KUKA KRL program: EPS_2_25089_SANMH03A_C_20251118074758.src

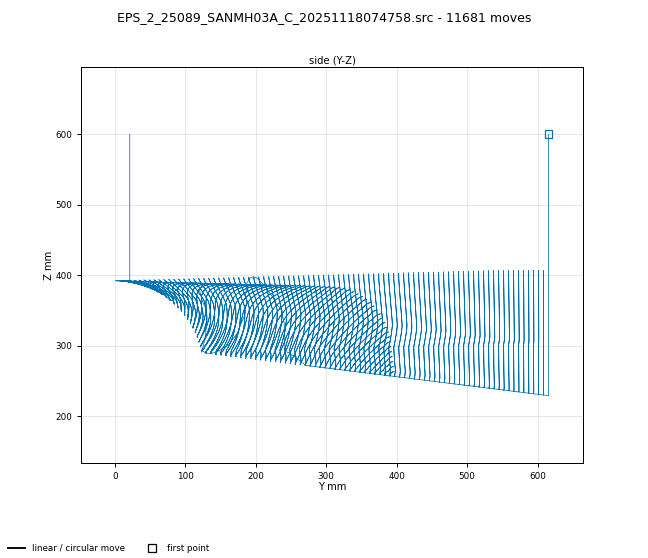
[picture p0: tool path of EPS_2_25089_SANMH03A_C_20251118074758.src, 11681 of 11683 moves have a stored position in this frame; points joined in program order, loops and branches not executed]
&ACCESS RVP
&REL 4
&COMMENT QRS 19112012
&PARAM EDITMASK = *
DEF PART()
EXT BAS (BAS_COMMAND :IN,REAL :IN )
INT I
BAS (#INITMOV,0 )

;KUKA QRS Post kuka4.cps  Date:22-06-2017 !

File_ID=2925

QRS_PRE_INIT()

;Init var - Until changes are made in qrs_pre_init
Outlet_Square_prg=0
Inlet_1_Square_prg=0
Inlet_2_Square_prg=0
Inlet_3_Square_prg=0
Inlet_4_Square_prg=0
Inlet_5_Square_prg=0

Outlet_1={X 0.000, Y 531.880, Z 306.500, B 0.000, E1 0.000 }
Inlet_1={X 0.000, Y 560.070, Z 281.500, B 0.000, E1 180.000 }
Outlet_1_type=201
Inlet_1_type=0
;QRS#1=Sidecore dimensions
;QRS#2=200-8" PVC SDR 35
;QRS#3=DeadEnd 201
;QRS#4=
;QRS#5=
;QRS#6=
;QRS#7=
;QRS#8=
;QRS#9=12-08 PSX
;QRS#10=

;QRS#11=
;QRS#12=
;QRS#13=
;QRS#14=
;QRS#15=
;QRS#16=1220x127x686 2,25'
;QRS#17=EPS Height
;QRS#18=407
;QRS#19=*
;QRS#20= UPDATED VERSION 22-06-2017
;QRS#21=*
Outlet_Square=0100
Inlet_1_Square=00
Inlet_2_Square=0
Inlet_3_Square=0
Inlet_4_Square=0
Inlet_5_Square=0
Mill_Square=1
Outlet_Square_Prg=204
Inlet_1_Square_prg=0

QRS_INIT()

$ADVANCE=5

; T1
PTP {E1 173.634,E2 173.634}
PTP {X 0,Y 615.433,A -85,B 0,C 180,E1 173.634,E2 173.634,E3 0,E4 0,E5 0,E6 0}
QRS_SPEED_INIT()
LIN {X 0,Y 615.433,Z 600,A -85,B 0,C 180,E1 173.634,E2 173.634,E3 0,E4 0,E5 0,E6 0} C_VEL
LIN {X 0,Y 615.433,Z 239.375,A -85,B 0,C 180,E1 173.634,E2 173.634} C_VEL
LIN {X 0,Y 615.433,Z 231.198,A -85,B 0,C 180,E1 173.634,E2 173.634} C_VEL
LIN {X 0,Y 615.441,Z 229.198,A -85,B 0,C 180,E1 173.448,E2 173.448} C_VEL
LIN {X 0,Y 615.497,Z 229.194,A -85,B 0,C 180,E1 170.806,E2 170.806} C_VEL
LIN {X 0,Y 615.433,Z 229.195,A -85,B 0,C 180,E1 168.143,E2 168.143} C_VEL
LIN {X 0,Y 615.431,Z 229.196,A -85,B 0,C 180,E1 166.083,E2 166.083} C_VEL
LIN {X 0,Y 615.468,Z 229.199,A -85,B 0,C 180,E1 163.418,E2 163.418} C_VEL
LIN {X 0,Y 615.454,Z 229.194,A -85,B 0,C 180,E1 160.666,E2 160.666} C_VEL
LIN {X 0,Y 615.441,Z 229.195,A -85,B 0,C 180,E1 158.572,E2 158.572} C_VEL
LIN {X 0,Y 615.432,Z 229.196,A -85,B 0,C 180,E1 156.447,E2 156.447} C_VEL
LIN {X 0,Y 615.428,Z 229.197,A -85,B 0,C 180,E1 154.288,E2 154.288} C_VEL
LIN {X 0,Y 615.484,Z 229.201,A -85,B 0,C 180,E1 151.548,E2 151.548} C_VEL
LIN {X 0,Y 615.446,Z 229.195,A -85,B 0,C 180,E1 148.918,E2 148.918} C_VEL
LIN {X 0,Y 615.426,Z 229.197,A -85,B 0,C 180,E1 146.472,E2 146.472} C_VEL
LIN {X 0,Y 615.44,Z 229.198,A -85,B 0,C 180,E1 144.17,E2 144.17} C_VEL
LIN {X 0,Y 615.468,Z 229.199,A -85,B 0,C 180,E1 141.938,E2 141.938} C_VEL
LIN {X 0,Y 615.468,Z 229.195,A -85,B 0,C 180,E1 139.4,E2 139.4} C_VEL
LIN {X 0,Y 615.427,Z 229.197,A -85,B 0,C 180,E1 136.957,E2 136.957} C_VEL
LIN {X 0,Y 615.424,Z 229.197,A -85,B 0,C 180,E1 134.935,E2 134.935} C_VEL
LIN {X 0,Y 615.448,Z 229.199,A -85,B 0,C 180,E1 132.355,E2 132.355} C_VEL
LIN {X 0,Y 615.475,Z 229.197,A -85,B 0,C 180,E1 129.75,E2 129.75} C_VEL
LIN {X 0,Y 615.426,Z 229.197,A -85,B 0,C 180,E1 127.245,E2 127.245} C_VEL
LIN {X 0,Y 615.434,Z 229.199,A -85,B 0,C 180,E1 124.705,E2 124.705} C_VEL
LIN {X 0,Y 615.478,Z 229.2,A -85,B 0,C 180,E1 122.342,E2 122.342} C_VEL
LIN {X 0,Y 615.45,Z 229.197,A -85,B 0,C 180,E1 119.802,E2 119.802} C_VEL
LIN {X 0,Y 615.452,Z 229.198,A -85,B 0,C 180,E1 117.916,E2 117.916} C_VEL
LIN {X 0,Y 615.423,Z 229.198,A -85,B 0,C 180,E1 115.572,E2 115.572} C_VEL
LIN {X 0,Y 615.419,Z 229.199,A -85,B 0,C 180,E1 113.559,E2 113.559} C_VEL
LIN {X 0,Y 615.416,Z 229.199,A -85,B 0,C 180,E1 111.434,E2 111.434} C_VEL
LIN {X 0,Y 615.419,Z 229.199,A -85,B 0,C 180,E1 109.34,E2 109.34} C_VEL
LIN {X 0,Y 615.474,Z 229.201,A -85,B 0,C 180,E1 106.452,E2 106.452} C_VEL
LIN {X 0,Y 615.419,Z 229.199,A -85,B 0,C 180,E1 103.875,E2 103.875} C_VEL
LIN {X 0,Y 615.415,Z 229.2,A -85,B 0,C 180,E1 101.862,E2 101.862} C_VEL
LIN {X 0,Y 615.416,Z 229.199,A -85,B 0,C 180,E1 99.863,E2 99.863} C_VEL
LIN {X 0,Y 615.414,Z 229.199,A -85,B 0,C 180,E1 97.876,E2 97.876} C_VEL
LIN {X 0,Y 615.414,Z 229.2,A -85,B 0,C 180,E1 95.899,E2 95.899} C_VEL
LIN {X 0,Y 615.449,Z 229.2,A -85,B 0,C 180,E1 93.273,E2 93.273} C_VEL
LIN {X 0,Y 615.452,Z 229.2,A -85,B 0,C 180,E1 90.654,E2 90.654} C_VEL
LIN {X 0,Y 615.412,Z 229.2,A -85,B 0,C 180,E1 88.037,E2 88.037} C_VEL
LIN {X 0,Y 615.457,Z 229.2,A -85,B 0,C 180,E1 85.415,E2 85.415} C_VEL
LIN {X 0,Y 615.445,Z 229.2,A -85,B 0,C 180,E1 82.784,E2 82.784} C_VEL
LIN {X 0,Y 615.416,Z 229.199,A -85,B 0,C 180,E1 80.137,E2 80.137} C_VEL
LIN {X 0,Y 615.477,Z 229.2,A -85,B 0,C 180,E1 77.47,E2 77.47} C_VEL
LIN {X 0,Y 615.428,Z 229.199,A -85,B 0,C 180,E1 74.773,E2 74.773} C_VEL
LIN {X 0,Y 615.423,Z 229.199,A -85,B 0,C 180,E1 72.728,E2 72.728} C_VEL
LIN {X 0,Y 615.419,Z 229.199,A -85,B 0,C 180,E1 70.66,E2 70.66} C_VEL
LIN {X 0,Y 615.416,Z 229.199,A -85,B 0,C 180,E1 68.566,E2 68.566} C_VEL
LIN {X 0,Y 615.419,Z 229.199,A -85,B 0,C 180,E1 66.442,E2 66.442} C_VEL
LIN {X 0,Y 615.484,Z 229.2,A -85,B 0,C 180,E1 63.556,E2 63.556} C_VEL
LIN {X 0,Y 615.45,Z 229.199,A -85,B 0,C 180,E1 61.341,E2 61.341} C_VEL
LIN {X 0,Y 615.42,Z 229.198,A -85,B 0,C 180,E1 58.911,E2 58.911} C_VEL
LIN {X 0,Y 615.434,Z 229.198,A -85,B 0,C 180,E1 56.461,E2 56.461} C_VEL
LIN {X 0,Y 615.455,Z 229.199,A -85,B 0,C 180,E1 53.574,E2 53.574} C_VEL
LIN {X 0,Y 615.422,Z 229.198,A -85,B 0,C 180,E1 50.935,E2 50.935} C_VEL
LIN {X 0,Y 615.451,Z 229.196,A -85,B 0,C 180,E1 48.524,E2 48.524} C_VEL
LIN {X 0,Y 615.465,Z 229.199,A -85,B 0,C 180,E1 45.85,E2 45.85} C_VEL
LIN {X 0,Y 615.479,Z 229.2,A -85,B 0,C 180,E1 43.998,E2 43.998} C_VEL
LIN {X 0,Y 615.427,Z 229.198,A -85,B 0,C 180,E1 41.471,E2 41.471} C_VEL
LIN {X 0,Y 615.442,Z 229.196,A -85,B 0,C 180,E1 38.9,E2 38.9} C_VEL
LIN {X 0,Y 615.482,Z 229.201,A -85,B 0,C 180,E1 36.418,E2 36.418} C_VEL
LIN {X 0,Y 615.452,Z 229.199,A -85,B 0,C 180,E1 34.017,E2 34.017} C_VEL
LIN {X 0,Y 615.428,Z 229.197,A -85,B 0,C 180,E1 31.682,E2 31.682} C_VEL
LIN {X 0,Y 615.428,Z 229.196,A -85,B 0,C 180,E1 29.403,E2 29.403} C_VEL
LIN {X 0,Y 615.457,Z 229.195,A -85,B 0,C 180,E1 27.042,E2 27.042} C_VEL
LIN {X 0,Y 615.454,Z 229.199,A -85,B 0,C 180,E1 24.268,E2 24.268} C_VEL
LIN {X 0,Y 615.439,Z 229.198,A -85,B 0,C 180,E1 22.133,E2 22.133} C_VEL
LIN {X 0,Y 615.432,Z 229.197,A -85,B 0,C 180,E1 20.029,E2 20.029} C_VEL
LIN {X 0,Y 615.43,Z 229.196,A -85,B 0,C 180,E1 17.953,E2 17.953} C_VEL
LIN {X 0,Y 615.48,Z 229.193,A -85,B 0,C 180,E1 15.221,E2 15.221} C_VEL
LIN {X 0,Y 615.451,Z 229.198,A -85,B 0,C 180,E1 12.526,E2 12.526} C_VEL
LIN {X 0,Y 615.447,Z 229.198,A -85,B 0,C 180,E1 10.523,E2 10.523} C_VEL
LIN {X 0,Y 615.445,Z 229.198,A -85,B 0,C 180,E1 8.533,E2 8.533} C_VEL
LIN {X 0,Y 615.444,Z 229.197,A -85,B 0,C 180,E1 6.553,E2 6.553} C_VEL
LIN {X 0,Y 615.443,Z 229.197,A -85,B 0,C 180,E1 4.581,E2 4.581} C_VEL
LIN {X 0,Y 615.441,Z 229.197,A -85,B 0,C 180,E1 2.614,E2 2.614} C_VEL
LIN {X 0,Y 615.441,Z 229.197,A -85,B 0,C 180,E1 0.65,E2 0.65} C_VEL
LIN {X 0,Y 615.441,Z 229.197,A -85,B 0,C 180,E1 -1.312,E2 -1.312} C_VEL
LIN {X 0,Y 615.441,Z 229.197,A -85,B 0,C 180,E1 -3.277,E2 -3.277} C_VEL
LIN {X 0,Y 615.44,Z 229.197,A -85,B 0,C 180,E1 -5.245,E2 -5.245} C_VEL
LIN {X 0,Y 615.44,Z 229.196,A -85,B 0,C 180,E1 -7.22,E2 -7.22} C_VEL
LIN {X 0,Y 615.439,Z 229.196,A -85,B 0,C 180,E1 -9.203,E2 -9.203} C_VEL
LIN {X 0,Y 615.438,Z 229.196,A -85,B 0,C 180,E1 -11.197,E2 -11.197} C_VEL
LIN {X 0,Y 615.469,Z 229.191,A -85,B 0,C 180,E1 -13.878,E2 -13.878} C_VEL
LIN {X 0,Y 615.468,Z 229.199,A -85,B 0,C 180,E1 -16.59,E2 -16.59} C_VEL
LIN {X 0,Y 615.457,Z 229.198,A -85,B 0,C 180,E1 -18.65,E2 -18.65} C_VEL
LIN {X 0,Y 615.449,Z 229.197,A -85,B 0,C 180,E1 -20.735,E2 -20.735} C_VEL
LIN {X 0,Y 615.442,Z 229.196,A -85,B 0,C 180,E1 -22.849,E2 -22.849} C_VEL
LIN {X 0,Y 615.439,Z 229.194,A -85,B 0,C 180,E1 -24.996,E2 -24.996} C_VEL
LIN {X 0,Y 615.496,Z 229.195,A -85,B 0,C 180,E1 -27.917,E2 -27.917} C_VEL
LIN {X 0,Y 615.481,Z 229.199,A -85,B 0,C 180,E1 -30.163,E2 -30.163} C_VEL
LIN {X 0,Y 615.45,Z 229.196,A -85,B 0,C 180,E1 -32.462,E2 -32.462} C_VEL
LIN {X 0,Y 615.439,Z 229.194,A -85,B 0,C 180,E1 -34.82,E2 -34.82} C_VEL
LIN {X 0,Y 615.473,Z 229.189,A -85,B 0,C 180,E1 -37.245,E2 -37.245} C_VEL
LIN {X 0,Y 615.464,Z 229.198,A -85,B 0,C 180,E1 -40.088,E2 -40.088} C_VEL
LIN {X 0,Y 615.444,Z 229.195,A -85,B 0,C 180,E1 -42.359,E2 -42.359} C_VEL
LIN {X 0,Y 615.471,Z 229.19,A -85,B 0,C 180,E1 -45.072,E2 -45.072} C_VEL
LIN {X 0,Y 615.468,Z 229.19,A -85,B 0,C 180,E1 -46.956,E2 -46.956} C_VEL
LIN {X 0,Y 615.491,Z 229.616,A -85,B 0,C 180,E1 -47.649,E2 -47.649} C_VEL
LIN {X 0,Y 615.439,Z 234.214,A -85,B 0,C 180,E1 -50.247,E2 -50.247} C_VEL
LIN {X 0,Y 615.494,Z 238.966,A -85,B 0,C 180,E1 -52.759,E2 -52.759} C_VEL
LIN {X 0,Y 615.486,Z 244.106,A -85,B 0,C 180,E1 -55.301,E2 -55.301} C_VEL
LIN {X 0,Y 615.472,Z 249.184,A -85,B 0,C 180,E1 -57.673,E2 -57.673} C_VEL
LIN {X 0,Y 615.449,Z 254.91,A -85,B 0,C 180,E1 -60.213,E2 -60.213} C_VEL
LIN {X 0,Y 615.475,Z 261.498,A -85,B 0,C 180,E1 -62.959,E2 -62.959} C_VEL
LIN {X 0,Y 615.47,Z 266.533,A -85,B 0,C 180,E1 -65.008,E2 -65.008} C_VEL
LIN {X 0,Y 615.475,Z 273.166,A -85,B 0,C 180,E1 -67.658,E2 -67.658} C_VEL
LIN {X 0,Y 615.484,Z 279.039,A -85,B 0,C 180,E1 -69.968,E2 -69.968} C_VEL
LIN {X 0,Y 615.488,Z 286.193,A -85,B 0,C 180,E1 -72.73,E2 -72.73} C_VEL
LIN {X 0,Y 615.466,Z 293.325,A -85,B 0,C 180,E1 -75.451,E2 -75.451} C_VEL
LIN {X 0,Y 615.478,Z 300.472,A -85,B 0,C 180,E1 -78.139,E2 -78.139} C_VEL
LIN {X 0,Y 615.498,Z 301.076,A -85,B 0,C 180,E1 -78.369,E2 -78.369} C_VEL
LIN {X 0,Y 615.485,Z 316.87,A -85,B 0,C 180,E1 -78.724,E2 -78.724} C_VEL
LIN {X 0,Y 615.445,Z 329.215,A -85,B 0,C 180,E1 -79.134,E2 -79.134} C_VEL
LIN {X 0,Y 615.44,Z 340.49,A -85,B 0,C 180,E1 -79.639,E2 -79.639} C_VEL
LIN {X 0,Y 615.49,Z 351.998,A -85,B 0,C 180,E1 -80.304,E2 -80.304} C_VEL
LIN {X 0,Y 615.499,Z 362.344,A -85,B 0,C 180,E1 -81.05,E2 -81.05} C_VEL
LIN {X 0,Y 615.497,Z 370.814,A -85,B 0,C 180,E1 -81.794,E2 -81.794} C_VEL
LIN {X 0,Y 615.498,Z 378.608,A -85,B 0,C 180,E1 -82.62,E2 -82.62} C_VEL
LIN {X 0,Y 615.496,Z 386.204,A -85,B 0,C 180,E1 -83.608,E2 -83.608} C_VEL
LIN {X 0,Y 615.498,Z 393.205,A -85,B 0,C 180,E1 -84.759,E2 -84.759} C_VEL
LIN {X 0,Y 615.494,Z 397.852,A -85,B 0,C 180,E1 -85.744,E2 -85.744} C_VEL
LIN {X 0,Y 615.494,Z 401.399,A -85,B 0,C 180,E1 -86.727,E2 -86.727} C_VEL
LIN {X 0,Y 615.497,Z 403.233,A -85,B 0,C 180,E1 -87.382,E2 -87.382} C_VEL
LIN {X 0,Y 615.5,Z 404.608,A -85,B 0,C 180,E1 -88.037,E2 -88.037} C_VEL
LIN {X 0,Y 615.496,Z 406.173,A -85,B 0,C 180,E1 -89.346,E2 -89.346} C_VEL
LIN {X 0,Y 615.494,Z 406.389,A -85,B 0,C 180,E1 -90,E2 -90} C_VEL
LIN {X 0,Y 615.495,Z 405.58,A -85,B 0,C 180,E1 -91.309,E2 -91.309} C_VEL
LIN {X 0,Y 615.5,Z 404.608,A -85,B 0,C 180,E1 -91.963,E2 -91.963} C_VEL
LIN {X 0,Y 615.497,Z 403.233,A -85,B 0,C 180,E1 -92.618,E2 -92.618} C_VEL
LIN {X 0,Y 615.496,Z 400.35,A -85,B 0,C 180,E1 -93.601,E2 -93.601} C_VEL
LIN {X 0,Y 615.498,Z 396.442,A -85,B 0,C 180,E1 -94.584,E2 -94.584} C_VEL
LIN {X 0,Y 615.499,Z 391.406,A -85,B 0,C 180,E1 -95.57,E2 -95.57} C_VEL
LIN {X 0,Y 615.497,Z 384.875,A -85,B 0,C 180,E1 -96.583,E2 -96.583} C_VEL
LIN {X 0,Y 615.497,Z 377.135,A -85,B 0,C 180,E1 -97.545,E2 -97.545} C_VEL
LIN {X 0,Y 615.498,Z 369.047,A -85,B 0,C 180,E1 -98.371,E2 -98.371} C_VEL
LIN {X 0,Y 615.499,Z 359.17,A -85,B 0,C 180,E1 -99.198,E2 -99.198} C_VEL
LIN {X 0,Y 615.472,Z 347.988,A -85,B 0,C 180,E1 -99.945,E2 -99.945} C_VEL
LIN {X 0,Y 615.437,Z 337.036,A -85,B 0,C 180,E1 -100.528,E2 -100.528} C_VEL
LIN {X 0,Y 615.457,Z 324.807,A -85,B 0,C 180,E1 -101.029,E2 -101.029} C_VEL
LIN {X 0,Y 615.499,Z 312.075,A -85,B 0,C 180,E1 -101.401,E2 -101.401} C_VEL
LIN {X 0,Y 615.498,Z 301.076,A -85,B 0,C 180,E1 -101.631,E2 -101.631} C_VEL
LIN {X 0,Y 615.471,Z 294.981,A -85,B 0,C 180,E1 -103.925,E2 -103.925} C_VEL
LIN {X 0,Y 615.486,Z 287.968,A -85,B 0,C 180,E1 -106.586,E2 -106.586} C_VEL
LIN {X 0,Y 615.484,Z 280.83,A -85,B 0,C 180,E1 -109.338,E2 -109.338} C_VEL
LIN {X 0,Y 615.494,Z 273.68,A -85,B 0,C 180,E1 -112.136,E2 -112.136} C_VEL
LIN {X 0,Y 615.467,Z 268.326,A -85,B 0,C 180,E1 -114.272,E2 -114.272} C_VEL
LIN {X 0,Y 615.446,Z 262.964,A -85,B 0,C 180,E1 -116.445,E2 -116.445} C_VEL
LIN {X 0,Y 615.48,Z 255.804,A -85,B 0,C 180,E1 -119.406,E2 -119.406} C_VEL
LIN {X 0,Y 615.454,Z 250.603,A -85,B 0,C 180,E1 -121.686,E2 -121.686} C_VEL
LIN {X 0,Y 615.484,Z 245.53,A -85,B 0,C 180,E1 -124.021,E2 -124.021} C_VEL
LIN {X 0,Y 615.469,Z 240.585,A -85,B 0,C 180,E1 -126.425,E2 -126.425} C_VEL
LIN {X 0,Y 615.499,Z 235.479,A -85,B 0,C 180,E1 -129.062,E2 -129.062} C_VEL
LIN {X 0,Y 615.447,Z 231.131,A -85,B 0,C 180,E1 -131.476,E2 -131.476} C_VEL
LIN {X 0,Y 615.491,Z 229.616,A -85,B 0,C 180,E1 -132.351,E2 -132.351} C_VEL
LIN {X 0,Y 615.452,Z 229.191,A -85,B 0,C 180,E1 -133.246,E2 -133.246} C_VEL
LIN {X 0,Y 615.462,Z 229.198,A -85,B 0,C 180,E1 -136.004,E2 -136.004} C_VEL
LIN {X 0,Y 615.469,Z 229.19,A -85,B 0,C 180,E1 -138.906,E2 -138.906} C_VEL
LIN {X 0,Y 615.449,Z 229.192,A -85,B 0,C 180,E1 -141.091,E2 -141.091} C_VEL
LIN {X 0,Y 615.447,Z 229.196,A -85,B 0,C 180,E1 -143.57,E2 -143.57} C_VEL
LIN {X 0,Y 615.493,Z 229.189,A -85,B 0,C 180,E1 -146.463,E2 -146.463} C_VEL
LIN {X 0,Y 615.441,Z 229.193,A -85,B 0,C 180,E1 -149.075,E2 -149.075} C_VEL
LIN {X 0,Y 615.457,Z 229.197,A -85,B 0,C 180,E1 -151.552,E2 -151.552} C_VEL
LIN {X 0,Y 615.472,Z 229.19,A -85,B 0,C 180,E1 -154.431,E2 -154.431} C_VEL
LIN {X 0,Y 615.465,Z 229.191,A -85,B 0,C 180,E1 -156.44,E2 -156.44} C_VEL
LIN {X 0,Y 615.45,Z 229.192,A -85,B 0,C 180,E1 -158.564,E2 -158.564} C_VEL
LIN {X 0,Y 615.441,Z 229.193,A -85,B 0,C 180,E1 -160.658,E2 -160.658} C_VEL
LIN {X 0,Y 615.437,Z 229.194,A -85,B 0,C 180,E1 -162.725,E2 -162.725} C_VEL
LIN {X 0,Y 615.48,Z 229.199,A -85,B 0,C 180,E1 -165.448,E2 -165.448} C_VEL
LIN {X 0,Y 615.463,Z 229.192,A -85,B 0,C 180,E1 -168.136,E2 -168.136} C_VEL
LIN {X 0,Y 615.457,Z 229.192,A -85,B 0,C 180,E1 -170.134,E2 -170.134} C_VEL
LIN {X 0,Y 615.454,Z 229.192,A -85,B 0,C 180,E1 -172.121,E2 -172.121} C_VEL
LIN {X 0,Y 615.451,Z 229.193,A -85,B 0,C 180,E1 -174.098,E2 -174.098} C_VEL
LIN {X 0,Y 615.449,Z 229.193,A -85,B 0,C 180,E1 -176.068,E2 -176.068} C_VEL
LIN {X 0,Y 615.447,Z 229.193,A -85,B 0,C 180,E1 -178.033,E2 -178.033} C_VEL
LIN {X 0,Y 615.446,Z 229.193,A -85,B 0,C 180,E1 -179.996,E2 -179.996} C_VEL
LIN {X 0,Y 615.444,Z 229.194,A -85,B 0,C 180,E1 -181.959,E2 -181.959} C_VEL
LIN {X 0,Y 615.443,Z 229.194,A -85,B 0,C 180,E1 -183.925,E2 -183.925} C_VEL
LIN {X 0,Y 615.441,Z 229.194,A -85,B 0,C 180,E1 -185.895,E2 -185.895} C_VEL
LIN {X 0,Y 615.441,Z 229.198,A -85,B 0,C 180,E1 -186.552,E2 -186.552} C_VEL
LIN {X 0,Y 614.816,Z 229.343,A -85,B 0,C 180,E1 -187.098,E2 -187.098} C_VEL
LIN {X 0,Y 612.019,Z 229.743,A -85,B 0,C 180,E1 -187.984,E2 -187.984} C_VEL
LIN {X 0,Y 609.616,Z 230.058,A -85,B 0,C 180,E1 -188.697,E2 -188.697} C_VEL
LIN {X 0,Y 608.553,Z 230.181,A -85,B 0,C 180,E1 -189.246,E2 -189.246} C_VEL
LIN {X 0,Y 608.45,Z 230.191,A -85,B 0,C 180,E1 -189.432,E2 -189.432} C_VEL
LIN {X 0,Y 608.416,Z 230.192,A -85,B 0,C 180,E1 -191.996,E2 -191.996} C_VEL
LIN {X 0,Y 608.452,Z 230.195,A -85,B 0,C 180,E1 -194.716,E2 -194.716} C_VEL
LIN {X 0,Y 608.422,Z 230.193,A -85,B 0,C 180,E1 -197.472,E2 -197.472} C_VEL
LIN {X 0,Y 608.413,Z 230.193,A -85,B 0,C 180,E1 -199.567,E2 -199.567} C_VEL
LIN {X 0,Y 608.424,Z 230.191,A -85,B 0,C 180,E1 -201.688,E2 -201.688} C_VEL
LIN {X 0,Y 608.428,Z 230.2,A -85,B 0,C 180,E1 -204.566,E2 -204.566} C_VEL
LIN {X 0,Y 608.407,Z 230.193,A -85,B 0,C 180,E1 -207.514,E2 -207.514} C_VEL
LIN {X 0,Y 608.419,Z 230.194,A -85,B 0,C 180,E1 -209.966,E2 -209.966} C_VEL
LIN {X 0,Y 608.429,Z 230.194,A -85,B 0,C 180,E1 -212.874,E2 -212.874} C_VEL
LIN {X 0,Y 608.399,Z 230.194,A -85,B 0,C 180,E1 -215.273,E2 -215.273} C_VEL
LIN {X 0,Y 608.441,Z 230.199,A -85,B 0,C 180,E1 -218.239,E2 -218.239} C_VEL
LIN {X 0,Y 608.464,Z 230.195,A -85,B 0,C 180,E1 -220.332,E2 -220.332} C_VEL
LIN {X 0,Y 608.402,Z 230.194,A -85,B 0,C 180,E1 -222.956,E2 -222.956} C_VEL
LIN {X 0,Y 608.399,Z 230.194,A -85,B 0,C 180,E1 -225.2,E2 -225.2} C_VEL
LIN {X 0,Y 608.454,Z 230.196,A -85,B 0,C 180,E1 -227.939,E2 -227.939} C_VEL
LIN {X 0,Y 608.424,Z 230.192,A -85,B 0,C 180,E1 -230.697,E2 -230.697} C_VEL
LIN {X 0,Y 608.393,Z 230.195,A -85,B 0,C 180,E1 -233.082,E2 -233.082} C_VEL
LIN {X 0,Y 608.433,Z 230.195,A -85,B 0,C 180,E1 -235.529,E2 -235.529} C_VEL
LIN {X 0,Y 608.443,Z 230.197,A -85,B 0,C 180,E1 -237.905,E2 -237.905} C_VEL
LIN {X 0,Y 608.432,Z 230.193,A -85,B 0,C 180,E1 -240.219,E2 -240.219} C_VEL
LIN {X 0,Y 608.412,Z 230.193,A -85,B 0,C 180,E1 -242.79,E2 -242.79} C_VEL
LIN {X 0,Y 608.45,Z 230.194,A -85,B 0,C 180,E1 -245.836,E2 -245.836} C_VEL
LIN {X 0,Y 608.415,Z 230.193,A -85,B 0,C 180,E1 -248.307,E2 -248.307} C_VEL
LIN {X 0,Y 608.435,Z 230.195,A -85,B 0,C 180,E1 -251.13,E2 -251.13} C_VEL
LIN {X 0,Y 608.416,Z 230.195,A -85,B 0,C 180,E1 -253.905,E2 -253.905} C_VEL
LIN {X 0,Y 608.401,Z 230.195,A -85,B 0,C 180,E1 -255.979,E2 -255.979} C_VEL
LIN {X 0,Y 608.402,Z 230.195,A -85,B 0,C 180,E1 -257.999,E2 -257.999} C_VEL
LIN {X 0,Y 608.395,Z 230.195,A -85,B 0,C 180,E1 -260.022,E2 -260.022} C_VEL
LIN {X 0,Y 608.412,Z 230.193,A -85,B 0,C 180,E1 -262.032,E2 -262.032} C_VEL
LIN {X 0,Y 608.422,Z 230.195,A -85,B 0,C 180,E1 -264.698,E2 -264.698} C_VEL
LIN {X 0,Y 608.442,Z 230.195,A -85,B 0,C 180,E1 -267.352,E2 -267.352} C_VEL
LIN {X 0,Y 608.403,Z 230.194,A -85,B 0,C 180,E1 -270,E2 -270} C_VEL
LIN {X 0,Y 608.442,Z 230.195,A -85,B 0,C 180,E1 -272.648,E2 -272.648} C_VEL
LIN {X 0,Y 608.422,Z 230.195,A -85,B 0,C 180,E1 -275.302,E2 -275.302} C_VEL
LIN {X 0,Y 608.412,Z 230.193,A -85,B 0,C 180,E1 -277.968,E2 -277.968} C_VEL
LIN {X 0,Y 608.444,Z 230.198,A -85,B 0,C 180,E1 -280.65,E2 -280.65} C_VEL
LIN {X 0,Y 608.405,Z 230.195,A -85,B 0,C 180,E1 -283.357,E2 -283.357} C_VEL
LIN {X 0,Y 608.411,Z 230.193,A -85,B 0,C 180,E1 -285.407,E2 -285.407} C_VEL
LIN {X 0,Y 608.391,Z 230.195,A -85,B 0,C 180,E1 -287.478,E2 -287.478} C_VEL
LIN {X 0,Y 608.392,Z 230.195,A -85,B 0,C 180,E1 -289.572,E2 -289.572} C_VEL
LIN {X 0,Y 608.48,Z 230.194,A -85,B 0,C 180,E1 -292.405,E2 -292.405} C_VEL
LIN {X 0,Y 608.42,Z 230.199,A -85,B 0,C 180,E1 -294.572,E2 -294.572} C_VEL
LIN {X 0,Y 608.412,Z 230.193,A -85,B 0,C 180,E1 -297.21,E2 -297.21} C_VEL
LIN {X 0,Y 608.464,Z 230.192,A -85,B 0,C 180,E1 -299.985,E2 -299.985} C_VEL
LIN {X 0,Y 608.407,Z 230.194,A -85,B 0,C 180,E1 -302.882,E2 -302.882} C_VEL
LIN {X 0,Y 608.396,Z 230.195,A -85,B 0,C 180,E1 -305.28,E2 -305.28} C_VEL
LIN {X 0,Y 608.444,Z 230.196,A -85,B 0,C 180,E1 -308.248,E2 -308.248} C_VEL
LIN {X 0,Y 608.425,Z 230.196,A -85,B 0,C 180,E1 -310.336,E2 -310.336} C_VEL
LIN {X 0,Y 608.395,Z 230.195,A -85,B 0,C 180,E1 -312.964,E2 -312.964} C_VEL
LIN {X 0,Y 608.452,Z 230.196,A -85,B 0,C 180,E1 -315.735,E2 -315.735} C_VEL
LIN {X 0,Y 608.459,Z 230.195,A -85,B 0,C 180,E1 -317.947,E2 -317.947} C_VEL
LIN {X 0,Y 608.397,Z 230.195,A -85,B 0,C 180,E1 -320.563,E2 -320.563} C_VEL
LIN {X 0,Y 608.416,Z 230.194,A -85,B 0,C 180,E1 -323.09,E2 -323.09} C_VEL
LIN {X 0,Y 608.45,Z 230.197,A -85,B 0,C 180,E1 -325.537,E2 -325.537} C_VEL
LIN {X 0,Y 608.444,Z 230.193,A -85,B 0,C 180,E1 -327.911,E2 -327.911} C_VEL
LIN {X 0,Y 608.414,Z 230.193,A -85,B 0,C 180,E1 -330.224,E2 -330.224} C_VEL
LIN {X 0,Y 608.441,Z 230.19,A -85,B 0,C 180,E1 -332.797,E2 -332.797} C_VEL
LIN {X 0,Y 608.435,Z 230.193,A -85,B 0,C 180,E1 -335.853,E2 -335.853} C_VEL
LIN {X 0,Y 608.424,Z 230.191,A -85,B 0,C 180,E1 -338.312,E2 -338.312} C_VEL
LIN {X 0,Y 608.434,Z 230.199,A -85,B 0,C 180,E1 -341.135,E2 -341.135} C_VEL
LIN {X 0,Y 608.414,Z 230.193,A -85,B 0,C 180,E1 -343.91,E2 -343.91} C_VEL
LIN {X 0,Y 608.451,Z 230.191,A -85,B 0,C 180,E1 -346.648,E2 -346.648} C_VEL
LIN {X 0,Y 608.438,Z 230.194,A -85,B 0,C 180,E1 -349.354,E2 -349.354} C_VEL
LIN {X 0,Y 608.425,Z 230.195,A -85,B 0,C 180,E1 -351.368,E2 -351.368} C_VEL
LIN {X 0,Y 608.42,Z 230.195,A -85,B 0,C 180,E1 -353.404,E2 -353.404} C_VEL
LIN {X 0,Y 608.415,Z 230.195,A -85,B 0,C 180,E1 -355.366,E2 -355.366} C_VEL
LIN {X 0,Y 608.437,Z 230.192,A -85,B 0,C 180,E1 -357.356,E2 -357.356} C_VEL
LIN {X 0,Y 608.439,Z 230.19,A -85,B 0,C 180,E1 -360.004,E2 -360.004} C_VEL
LIN {X 0,Y 608.48,Z 230.194,A -85,B 0,C 180,E1 -362.652,E2 -362.652} C_VEL
LIN {X 0,Y 608.423,Z 230.192,A -85,B 0,C 180,E1 -365.306,E2 -365.306} C_VEL
LIN {X 0,Y 608.413,Z 230.193,A -85,B 0,C 180,E1 -367.303,E2 -367.303} C_VEL
LIN {X 0,Y 608.434,Z 230.192,A -85,B 0,C 180,E1 -369.981,E2 -369.981} C_VEL
LIN {X 0,Y 608.461,Z 230.193,A -85,B 0,C 180,E1 -372.68,E2 -372.68} C_VEL
LIN {X 0,Y 608.437,Z 230.189,A -85,B 0,C 180,E1 -375.41,E2 -375.41} C_VEL
LIN {X 0,Y 608.443,Z 230.197,A -85,B 0,C 180,E1 -378.175,E2 -378.175} C_VEL
LIN {X 0,Y 608.428,Z 230.191,A -85,B 0,C 180,E1 -380.985,E2 -380.985} C_VEL
LIN {X 0,Y 608.42,Z 230.192,A -85,B 0,C 180,E1 -383.128,E2 -383.128} C_VEL
LIN {X 0,Y 608.469,Z 230.189,A -85,B 0,C 180,E1 -385.723,E2 -385.723} C_VEL
LIN {X 0,Y 608.443,Z 230.191,A -85,B 0,C 180,E1 -388.617,E2 -388.617} C_VEL
LIN {X 0,Y 608.429,Z 230.193,A -85,B 0,C 180,E1 -390.55,E2 -390.55} C_VEL
LIN {X 0,Y 608.433,Z 230.19,A -85,B 0,C 180,E1 -392.883,E2 -392.883} C_VEL
LIN {X 0,Y 608.432,Z 230.192,A -85,B 0,C 180,E1 -395.281,E2 -395.281} C_VEL
LIN {X 0,Y 608.457,Z 230.196,A -85,B 0,C 180,E1 -397.749,E2 -397.749} C_VEL
LIN {X 0,Y 608.435,Z 230.192,A -85,B 0,C 180,E1 -400.329,E2 -400.329} C_VEL
LIN {X 0,Y 608.479,Z 230.189,A -85,B 0,C 180,E1 -403.311,E2 -403.311} C_VEL
LIN {X 0,Y 608.446,Z 230.192,A -85,B 0,C 180,E1 -406.13,E2 -406.13} C_VEL
LIN {X 0,Y 608.435,Z 230.193,A -85,B 0,C 180,E1 -407.04,E2 -407.04} C_VEL
LIN {X 0,Y 608.477,Z 231.423,A -85,B 0,C 180,E1 -407.941,E2 -407.941} C_VEL
LIN {X 0,Y 608.501,Z 236.288,A -85,B 0,C 180,E1 -410.701,E2 -410.701} C_VEL
LIN {X 0,Y 608.514,Z 240.828,A -85,B 0,C 180,E1 -413.09,E2 -413.09} C_VEL
LIN {X 0,Y 608.469,Z 245.748,A -85,B 0,C 180,E1 -415.532,E2 -415.532} C_VEL
LIN {X 0,Y 608.449,Z 250.809,A -85,B 0,C 180,E1 -417.905,E2 -417.905} C_VEL
LIN {X 0,Y 608.436,Z 255.969,A -85,B 0,C 180,E1 -420.22,E2 -420.22} C_VEL
LIN {X 0,Y 608.417,Z 263.124,A -85,B 0,C 180,E1 -423.225,E2 -423.225} C_VEL
LIN {X 0,Y 608.439,Z 268.514,A -85,B 0,C 180,E1 -425.429,E2 -425.429} C_VEL
LIN {X 0,Y 608.453,Z 275.699,A -85,B 0,C 180,E1 -428.308,E2 -428.308} C_VEL
LIN {X 0,Y 608.457,Z 283.293,A -85,B 0,C 180,E1 -431.29,E2 -431.29} C_VEL
LIN {X 0,Y 608.434,Z 290.071,A -85,B 0,C 180,E1 -433.906,E2 -433.906} C_VEL
LIN {X 0,Y 608.432,Z 297.257,A -85,B 0,C 180,E1 -436.643,E2 -436.643} C_VEL
LIN {X 0,Y 608.459,Z 301.63,A -85,B 0,C 180,E1 -438.254,E2 -438.254} C_VEL
LIN {X 0,Y 608.546,Z 314.714,A -85,B 0,C 180,E1 -438.53,E2 -438.53} C_VEL
LIN {X 0,Y 608.475,Z 327.56,A -85,B 0,C 180,E1 -438.941,E2 -438.941} C_VEL
LIN {X 0,Y 608.467,Z 338.929,A -85,B 0,C 180,E1 -439.435,E2 -439.435} C_VEL
LIN {X 0,Y 608.471,Z 349.582,A -85,B 0,C 180,E1 -440.023,E2 -440.023} C_VEL
LIN {X 0,Y 608.483,Z 360.478,A -85,B 0,C 180,E1 -440.778,E2 -440.778} C_VEL
LIN {X 0,Y 608.475,Z 371.115,A -85,B 0,C 180,E1 -441.699,E2 -441.699} C_VEL
LIN {X 0,Y 608.471,Z 378.961,A -85,B 0,C 180,E1 -442.534,E2 -442.534} C_VEL
LIN {X 0,Y 608.461,Z 386.29,A -85,B 0,C 180,E1 -443.485,E2 -443.485} C_VEL
LIN {X 0,Y 608.451,Z 391.865,A -85,B 0,C 180,E1 -444.366,E2 -444.366} C_VEL
LIN {X 0,Y 608.432,Z 396.951,A -85,B 0,C 180,E1 -445.362,E2 -445.362} C_VEL
LIN {X 0,Y 608.449,Z 400.896,A -85,B 0,C 180,E1 -446.358,E2 -446.358} C_VEL
LIN {X 0,Y 608.425,Z 403.808,A -85,B 0,C 180,E1 -447.352,E2 -447.352} C_VEL
LIN {X 0,Y 608.445,Z 405.201,A -85,B 0,C 180,E1 -448.014,E2 -448.014} C_VEL
LIN {X 0,Y 608.439,Z 406.783,A -85,B 0,C 180,E1 -449.338,E2 -449.338} C_VEL
LIN {X 0,Y 608.434,Z 406.998,A -85,B 0,C 180,E1 -450,E2 -450} C_VEL
LIN {X 0,Y 608.448,Z 406.184,A -85,B 0,C 180,E1 -451.324,E2 -451.324} C_VEL
LIN {X 0,Y 608.445,Z 405.201,A -85,B 0,C 180,E1 -451.986,E2 -451.986} C_VEL
LIN {X 0,Y 608.425,Z 403.808,A -85,B 0,C 180,E1 -452.648,E2 -452.648} C_VEL
LIN {X 0,Y 608.449,Z 400.896,A -85,B 0,C 180,E1 -453.642,E2 -453.642} C_VEL
LIN {X 0,Y 608.432,Z 396.951,A -85,B 0,C 180,E1 -454.638,E2 -454.638} C_VEL
LIN {X 0,Y 608.451,Z 391.865,A -85,B 0,C 180,E1 -455.634,E2 -455.634} C_VEL
LIN {X 0,Y 608.442,Z 385.473,A -85,B 0,C 180,E1 -456.633,E2 -456.633} C_VEL
LIN {X 0,Y 608.476,Z 377.48,A -85,B 0,C 180,E1 -457.633,E2 -457.633} C_VEL
LIN {X 0,Y 608.487,Z 369.34,A -85,B 0,C 180,E1 -458.468,E2 -458.468} C_VEL
LIN {X 0,Y 608.487,Z 359.4,A -85,B 0,C 180,E1 -459.305,E2 -459.305} C_VEL
LIN {X 0,Y 608.48,Z 348.171,A -85,B 0,C 180,E1 -460.061,E2 -460.061} C_VEL
LIN {X 0,Y 608.463,Z 335.887,A -85,B 0,C 180,E1 -460.712,E2 -460.712} C_VEL
LIN {X 0,Y 608.492,Z 324.097,A -85,B 0,C 180,E1 -461.186,E2 -461.186} C_VEL
LIN {X 0,Y 608.551,Z 311.272,A -85,B 0,C 180,E1 -461.554,E2 -461.554} C_VEL
LIN {X 0,Y 608.436,Z 301.468,A -85,B 0,C 180,E1 -461.768,E2 -461.768} C_VEL
LIN {X 0,Y 608.432,Z 293.664,A -85,B 0,C 180,E1 -464.721,E2 -464.721} C_VEL
LIN {X 0,Y 608.431,Z 286.478,A -85,B 0,C 180,E1 -467.477,E2 -467.477} C_VEL
LIN {X 0,Y 608.451,Z 281.089,A -85,B 0,C 180,E1 -469.57,E2 -469.57} C_VEL
LIN {X 0,Y 608.433,Z 273.747,A -85,B 0,C 180,E1 -472.469,E2 -472.469} C_VEL
LIN {X 0,Y 608.439,Z 268.514,A -85,B 0,C 180,E1 -474.571,E2 -474.571} C_VEL
LIN {X 0,Y 608.455,Z 262.089,A -85,B 0,C 180,E1 -477.201,E2 -477.201} C_VEL
LIN {X 0,Y 608.431,Z 255.559,A -85,B 0,C 180,E1 -479.964,E2 -479.964} C_VEL
LIN {X 0,Y 608.483,Z 249.869,A -85,B 0,C 180,E1 -482.524,E2 -482.524} C_VEL
LIN {X 0,Y 608.477,Z 244.098,A -85,B 0,C 180,E1 -485.274,E2 -485.274} C_VEL
LIN {X 0,Y 608.475,Z 239.204,A -85,B 0,C 180,E1 -487.745,E2 -487.745} C_VEL
LIN {X 0,Y 608.458,Z 234.44,A -85,B 0,C 180,E1 -490.328,E2 -490.328} C_VEL
LIN {X 0,Y 608.506,Z 230.938,A -85,B 0,C 180,E1 -492.337,E2 -492.337} C_VEL
LIN {X 0,Y 608.435,Z 230.194,A -85,B 0,C 180,E1 -492.96,E2 -492.96} C_VEL
LIN {X 0,Y 608.426,Z 230.193,A -85,B 0,C 180,E1 -495.738,E2 -495.738} C_VEL
LIN {X 0,Y 608.439,Z 230.194,A -85,B 0,C 180,E1 -497.935,E2 -497.935} C_VEL
LIN {X 0,Y 608.433,Z 230.193,A -85,B 0,C 180,E1 -500.705,E2 -500.705} C_VEL
LIN {X 0,Y 608.419,Z 230.192,A -85,B 0,C 180,E1 -503.08,E2 -503.08} C_VEL
LIN {X 0,Y 608.439,Z 230.191,A -85,B 0,C 180,E1 -505.526,E2 -505.526} C_VEL
LIN {X 0,Y 608.451,Z 230.196,A -85,B 0,C 180,E1 -507.902,E2 -507.902} C_VEL
LIN {X 0,Y 608.48,Z 230.19,A -85,B 0,C 180,E1 -510.219,E2 -510.219} C_VEL
LIN {X 0,Y 608.412,Z 230.194,A -85,B 0,C 180,E1 -513.221,E2 -513.221} C_VEL
LIN {X 0,Y 608.481,Z 230.195,A -85,B 0,C 180,E1 -515.844,E2 -515.844} C_VEL
LIN {X 0,Y 608.451,Z 230.19,A -85,B 0,C 180,E1 -518.305,E2 -518.305} C_VEL
LIN {X 0,Y 608.433,Z 230.192,A -85,B 0,C 180,E1 -521.127,E2 -521.127} C_VEL
LIN {X 0,Y 608.458,Z 230.193,A -85,B 0,C 180,E1 -523.903,E2 -523.903} C_VEL
LIN {X 0,Y 608.425,Z 230.191,A -85,B 0,C 180,E1 -526.64,E2 -526.64} C_VEL
LIN {X 0,Y 608.454,Z 230.195,A -85,B 0,C 180,E1 -529.347,E2 -529.347} C_VEL
LIN {X 0,Y 608.425,Z 230.193,A -85,B 0,C 180,E1 -532.029,E2 -532.029} C_VEL
LIN {X 0,Y 608.43,Z 230.192,A -85,B 0,C 180,E1 -534.029,E2 -534.029} C_VEL
LIN {X 0,Y 608.421,Z 230.193,A -85,B 0,C 180,E1 -536.022,E2 -536.022} C_VEL
LIN {X 0,Y 608.42,Z 230.192,A -85,B 0,C 180,E1 -538.01,E2 -538.01} C_VEL
LIN {X 0,Y 608.439,Z 230.19,A -85,B 0,C 180,E1 -539.996,E2 -539.996} C_VEL
LIN {X 0,Y 608.437,Z 230.192,A -85,B 0,C 180,E1 -542.644,E2 -542.644} C_VEL
LIN {X 0,Y 608.468,Z 230.193,A -85,B 0,C 180,E1 -545.298,E2 -545.298} C_VEL
LIN {X 0,Y 608.407,Z 230.193,A -85,B 0,C 180,E1 -547.963,E2 -547.963} C_VEL
LIN {X 0,Y 608.45,Z 230.191,A -85,B 0,C 180,E1 -549.432,E2 -549.432} C_VEL
LIN {X 0,Y 607.741,Z 230.279,A -85,B 0,C 180,E1 -549.985,E2 -549.985} C_VEL
LIN {X 0,Y 604.87,Z 230.643,A -85,B 0,C 180,E1 -550.882,E2 -550.882} C_VEL
LIN {X 0,Y 602.475,Z 230.936,A -85,B 0,C 180,E1 -551.604,E2 -551.604} C_VEL
LIN {X 0,Y 601.455,Z 231.06,A -85,B 0,C 180,E1 -552.16,E2 -552.16} C_VEL
LIN {X 0,Y 601.376,Z 231.071,A -85,B 0,C 180,E1 -552.349,E2 -552.349} C_VEL
LIN {X 0,Y 601.407,Z 231.075,A -85,B 0,C 180,E1 -554.892,E2 -554.892} C_VEL
LIN {X 0,Y 601.407,Z 231.073,A -85,B 0,C 180,E1 -556.981,E2 -556.981} C_VEL
LIN {X 0,Y 601.37,Z 231.07,A -85,B 0,C 180,E1 -559.805,E2 -559.805} C_VEL
LIN {X 0,Y 601.376,Z 231.07,A -85,B 0,C 180,E1 -561.955,E2 -561.955} C_VEL
LIN {X 0,Y 601.397,Z 231.071,A -85,B 0,C 180,E1 -564.287,E2 -564.287} C_VEL
LIN {X 0,Y 601.419,Z 231.066,A -85,B 0,C 180,E1 -567.106,E2 -567.106} C_VEL
LIN {X 0,Y 601.377,Z 231.069,A -85,B 0,C 180,E1 -569.389,E2 -569.389} C_VEL
LIN {X 0,Y 601.427,Z 231.072,A -85,B 0,C 180,E1 -572.509,E2 -572.509} C_VEL
LIN {X 0,Y 601.374,Z 231.07,A -85,B 0,C 180,E1 -575.111,E2 -575.111} C_VEL
LIN {X 0,Y 601.389,Z 231.068,A -85,B 0,C 180,E1 -577.415,E2 -577.415} C_VEL
LIN {X 0,Y 601.389,Z 231.074,A -85,B 0,C 180,E1 -579.989,E2 -579.989} C_VEL
LIN {X 0,Y 601.402,Z 231.069,A -85,B 0,C 180,E1 -582.663,E2 -582.663} C_VEL
LIN {X 0,Y 601.372,Z 231.071,A -85,B 0,C 180,E1 -585.478,E2 -585.478} C_VEL
LIN {X 0,Y 601.384,Z 231.072,A -85,B 0,C 180,E1 -588.401,E2 -588.401} C_VEL
LIN {X 0,Y 601.384,Z 231.068,A -85,B 0,C 180,E1 -590.872,E2 -590.872} C_VEL
LIN {X 0,Y 601.393,Z 231.074,A -85,B 0,C 180,E1 -593.729,E2 -593.729} C_VEL
LIN {X 0,Y 601.382,Z 231.068,A -85,B 0,C 180,E1 -596.685,E2 -596.685} C_VEL
LIN {X 0,Y 601.433,Z 231.071,A -85,B 0,C 180,E1 -599.837,E2 -599.837} C_VEL
LIN {X 0,Y 601.356,Z 231.072,A -85,B 0,C 180,E1 -602.633,E2 -602.633} C_VEL
LIN {X 0,Y 601.355,Z 231.074,A -85,B 0,C 180,E1 -605.12,E2 -605.12} C_VEL
LIN {X 0,Y 601.402,Z 231.073,A -85,B 0,C 180,E1 -607.379,E2 -607.379} C_VEL
LIN {X 0,Y 601.357,Z 231.072,A -85,B 0,C 180,E1 -610.189,E2 -610.189} C_VEL
LIN {X 0,Y 601.381,Z 231.072,A -85,B 0,C 180,E1 -613.013,E2 -613.013} C_VEL
LIN {X 0,Y 601.354,Z 231.074,A -85,B 0,C 180,E1 -615.904,E2 -615.904} C_VEL
LIN {X 0,Y 601.364,Z 231.073,A -85,B 0,C 180,E1 -617.857,E2 -617.857} C_VEL
LIN {X 0,Y 601.379,Z 231.07,A -85,B 0,C 180,E1 -619.904,E2 -619.904} C_VEL
LIN {X 0,Y 601.391,Z 231.069,A -85,B 0,C 180,E1 -622.614,E2 -622.614} C_VEL
LIN {X 0,Y 601.389,Z 231.075,A -85,B 0,C 180,E1 -625.308,E2 -625.308} C_VEL
LIN {X 0,Y 601.354,Z 231.072,A -85,B 0,C 180,E1 -627.991,E2 -627.991} C_VEL
LIN {X 0,Y 601.41,Z 231.07,A -85,B 0,C 180,E1 -630.67,E2 -630.67} C_VEL
LIN {X 0,Y 601.387,Z 231.072,A -85,B 0,C 180,E1 -633.35,E2 -633.35} C_VEL
LIN {X 0,Y 601.349,Z 231.073,A -85,B 0,C 180,E1 -636.038,E2 -636.038} C_VEL
LIN {X 0,Y 601.414,Z 231.074,A -85,B 0,C 180,E1 -638.738,E2 -638.738} C_VEL
LIN {X 0,Y 601.371,Z 231.071,A -85,B 0,C 180,E1 -641.459,E2 -641.459} C_VEL
LIN {X 0,Y 601.355,Z 231.072,A -85,B 0,C 180,E1 -643.517,E2 -643.517} C_VEL
LIN {X 0,Y 601.408,Z 231.07,A -85,B 0,C 180,E1 -646.287,E2 -646.287} C_VEL
LIN {X 0,Y 601.374,Z 231.071,A -85,B 0,C 180,E1 -649.1,E2 -649.1} C_VEL
LIN {X 0,Y 601.354,Z 231.072,A -85,B 0,C 180,E1 -651.241,E2 -651.241} C_VEL
LIN {X 0,Y 601.368,Z 231.07,A -85,B 0,C 180,E1 -653.412,E2 -653.412} C_VEL
LIN {X 0,Y 601.366,Z 231.073,A -85,B 0,C 180,E1 -655.874,E2 -655.874} C_VEL
LIN {X 0,Y 601.398,Z 231.071,A -85,B 0,C 180,E1 -658.628,E2 -658.628} C_VEL
LIN {X 0,Y 601.38,Z 231.069,A -85,B 0,C 180,E1 -660.943,E2 -660.943} C_VEL
LIN {X 0,Y 601.383,Z 231.068,A -85,B 0,C 180,E1 -663.315,E2 -663.315} C_VEL
LIN {X 0,Y 601.393,Z 231.074,A -85,B 0,C 180,E1 -666.271,E2 -666.271} C_VEL
LIN {X 0,Y 601.384,Z 231.068,A -85,B 0,C 180,E1 -669.128,E2 -669.128} C_VEL
LIN {X 0,Y 601.392,Z 231.074,A -85,B 0,C 180,E1 -671.767,E2 -671.767} C_VEL
LIN {X 0,Y 601.37,Z 231.071,A -85,B 0,C 180,E1 -674.539,E2 -674.539} C_VEL
LIN {X 0,Y 601.411,Z 231.068,A -85,B 0,C 180,E1 -677.408,E2 -677.408} C_VEL
LIN {X 0,Y 601.389,Z 231.074,A -85,B 0,C 180,E1 -680.011,E2 -680.011} C_VEL
LIN {X 0,Y 601.389,Z 231.067,A -85,B 0,C 180,E1 -682.622,E2 -682.622} C_VEL
LIN {X 0,Y 601.403,Z 231.068,A -85,B 0,C 180,E1 -685.075,E2 -685.075} C_VEL
LIN {X 0,Y 601.427,Z 231.072,A -85,B 0,C 180,E1 -687.491,E2 -687.491} C_VEL
LIN {X 0,Y 601.377,Z 231.069,A -85,B 0,C 180,E1 -690.611,E2 -690.611} C_VEL
LIN {X 0,Y 601.417,Z 231.066,A -85,B 0,C 180,E1 -692.893,E2 -692.893} C_VEL
LIN {X 0,Y 601.414,Z 231.067,A -85,B 0,C 180,E1 -695.864,E2 -695.864} C_VEL
LIN {X 0,Y 601.379,Z 231.071,A -85,B 0,C 180,E1 -698.765,E2 -698.765} C_VEL
LIN {X 0,Y 601.373,Z 231.073,A -85,B 0,C 180,E1 -701.612,E2 -701.612} C_VEL
LIN {X 0,Y 601.4,Z 231.068,A -85,B 0,C 180,E1 -703.717,E2 -703.717} C_VEL
LIN {X 0,Y 601.391,Z 231.069,A -85,B 0,C 180,E1 -706.488,E2 -706.488} C_VEL
LIN {X 0,Y 601.406,Z 231.072,A -85,B 0,C 180,E1 -709.228,E2 -709.228} C_VEL
LIN {X 0,Y 601.382,Z 231.068,A -85,B 0,C 180,E1 -711.943,E2 -711.943} C_VEL
LIN {X 0,Y 601.426,Z 231.069,A -85,B 0,C 180,E1 -714.64,E2 -714.64} C_VEL
LIN {X 0,Y 601.406,Z 231.068,A -85,B 0,C 180,E1 -717.325,E2 -717.325} C_VEL
LIN {X 0,Y 601.41,Z 231.065,A -85,B 0,C 180,E1 -720.004,E2 -720.004} C_VEL
LIN {X 0,Y 601.441,Z 231.072,A -85,B 0,C 180,E1 -722.683,E2 -722.683} C_VEL
LIN {X 0,Y 601.389,Z 231.068,A -85,B 0,C 180,E1 -725.368,E2 -725.368} C_VEL
LIN {X 0,Y 601.399,Z 231.069,A -85,B 0,C 180,E1 -728.065,E2 -728.065} C_VEL
LIN {X 0,Y 601.398,Z 231.069,A -85,B 0,C 180,E1 -731.006,E2 -731.006} C_VEL
LIN {X 0,Y 601.389,Z 231.068,A -85,B 0,C 180,E1 -733.52,E2 -733.52} C_VEL
LIN {X 0,Y 601.426,Z 231.072,A -85,B 0,C 180,E1 -736.29,E2 -736.29} C_VEL
LIN {X 0,Y 601.4,Z 231.066,A -85,B 0,C 180,E1 -739.102,E2 -739.102} C_VEL
LIN {X 0,Y 601.387,Z 231.068,A -85,B 0,C 180,E1 -741.243,E2 -741.243} C_VEL
LIN {X 0,Y 601.459,Z 231.069,A -85,B 0,C 180,E1 -744.143,E2 -744.143} C_VEL
LIN {X 0,Y 601.383,Z 231.068,A -85,B 0,C 180,E1 -747.117,E2 -747.117} C_VEL
LIN {X 0,Y 601.4,Z 231.068,A -85,B 0,C 180,E1 -749.397,E2 -749.397} C_VEL
LIN {X 0,Y 601.393,Z 231.073,A -85,B 0,C 180,E1 -751.73,E2 -751.73} C_VEL
LIN {X 0,Y 601.418,Z 231.071,A -85,B 0,C 180,E1 -754.121,E2 -754.121} C_VEL
LIN {X 0,Y 601.383,Z 231.069,A -85,B 0,C 180,E1 -756.587,E2 -756.587} C_VEL
LIN {X 0,Y 601.394,Z 231.068,A -85,B 0,C 180,E1 -759.13,E2 -759.13} C_VEL
LIN {X 0,Y 601.413,Z 231.075,A -85,B 0,C 180,E1 -761.768,E2 -761.768} C_VEL
LIN {X 0,Y 601.401,Z 231.067,A -85,B 0,C 180,E1 -764.534,E2 -764.534} C_VEL
LIN {X 0,Y 601.405,Z 231.069,A -85,B 0,C 180,E1 -766.432,E2 -766.432} C_VEL
LIN {X 0,Y 601.488,Z 231.795,A -85,B 0,C 180,E1 -767.403,E2 -767.403} C_VEL
LIN {X 0,Y 601.459,Z 236.268,A -85,B 0,C 180,E1 -770.01,E2 -770.01} C_VEL
LIN {X 0,Y 601.485,Z 241.07,A -85,B 0,C 180,E1 -772.614,E2 -772.614} C_VEL
LIN {X 0,Y 601.464,Z 245.9,A -85,B 0,C 180,E1 -775.072,E2 -775.072} C_VEL
LIN {X 0,Y 601.455,Z 250.931,A -85,B 0,C 180,E1 -777.487,E2 -777.487} C_VEL
LIN {X 0,Y 601.404,Z 256.113,A -85,B 0,C 180,E1 -779.857,E2 -779.857} C_VEL
LIN {X 0,Y 601.397,Z 262.541,A -85,B 0,C 180,E1 -782.643,E2 -782.643} C_VEL
LIN {X 0,Y 601.391,Z 268.514,A -85,B 0,C 180,E1 -785.122,E2 -785.122} C_VEL
LIN {X 0,Y 601.369,Z 274.129,A -85,B 0,C 180,E1 -787.407,E2 -787.407} C_VEL
LIN {X 0,Y 601.378,Z 281.089,A -85,B 0,C 180,E1 -790.19,E2 -790.19} C_VEL
LIN {X 0,Y 601.358,Z 288.275,A -85,B 0,C 180,E1 -793.012,E2 -793.012} C_VEL
LIN {X 0,Y 601.352,Z 295.834,A -85,B 0,C 180,E1 -795.937,E2 -795.937} C_VEL
LIN {X 0,Y 601.37,Z 301.586,A -85,B 0,C 180,E1 -798.114,E2 -798.114} C_VEL
LIN {X 0,Y 601.609,Z 311.263,A -85,B 0,C 180,E1 -798.311,E2 -798.311} C_VEL
LIN {X 0,Y 601.537,Z 323.222,A -85,B 0,C 180,E1 -798.655,E2 -798.655} C_VEL
LIN {X 0,Y 601.48,Z 335.279,A -85,B 0,C 180,E1 -799.134,E2 -799.134} C_VEL
LIN {X 0,Y 601.473,Z 346.76,A -85,B 0,C 180,E1 -799.736,E2 -799.736} C_VEL
LIN {X 0,Y 601.462,Z 358.25,A -85,B 0,C 180,E1 -800.5,E2 -800.5} C_VEL
LIN {X 0,Y 601.436,Z 367.522,A -85,B 0,C 180,E1 -801.263,E2 -801.263} C_VEL
LIN {X 0,Y 601.401,Z 375.996,A -85,B 0,C 180,E1 -802.108,E2 -802.108} C_VEL
LIN {X 0,Y 601.383,Z 384.24,A -85,B 0,C 180,E1 -803.12,E2 -803.12} C_VEL
LIN {X 0,Y 601.361,Z 389.869,A -85,B 0,C 180,E1 -803.963,E2 -803.963} C_VEL
LIN {X 0,Y 601.345,Z 395.365,A -85,B 0,C 180,E1 -804.971,E2 -804.971} C_VEL
LIN {X 0,Y 601.347,Z 399.672,A -85,B 0,C 180,E1 -805.979,E2 -805.979} C_VEL
LIN {X 0,Y 601.344,Z 401.959,A -85,B 0,C 180,E1 -806.65,E2 -806.65} C_VEL
LIN {X 0,Y 601.325,Z 403.805,A -85,B 0,C 180,E1 -807.321,E2 -807.321} C_VEL
LIN {X 0,Y 601.343,Z 405.199,A -85,B 0,C 180,E1 -807.991,E2 -807.991} C_VEL
LIN {X 0,Y 601.339,Z 406.783,A -85,B 0,C 180,E1 -809.33,E2 -809.33} C_VEL
LIN {X 0,Y 601.335,Z 406.99,A -85,B 0,C 180,E1 -810,E2 -810} C_VEL
LIN {X 0,Y 601.348,Z 406.186,A -85,B 0,C 180,E1 -811.339,E2 -811.339} C_VEL
LIN {X 0,Y 601.343,Z 405.199,A -85,B 0,C 180,E1 -812.009,E2 -812.009} C_VEL
LIN {X 0,Y 601.325,Z 403.805,A -85,B 0,C 180,E1 -812.679,E2 -812.679} C_VEL
LIN {X 0,Y 601.368,Z 400.894,A -85,B 0,C 180,E1 -813.685,E2 -813.685} C_VEL
LIN {X 0,Y 601.336,Z 396.949,A -85,B 0,C 180,E1 -814.693,E2 -814.693} C_VEL
LIN {X 0,Y 601.374,Z 391.857,A -85,B 0,C 180,E1 -815.701,E2 -815.701} C_VEL
LIN {X 0,Y 601.383,Z 385.471,A -85,B 0,C 180,E1 -816.711,E2 -816.711} C_VEL
LIN {X 0,Y 601.396,Z 377.484,A -85,B 0,C 180,E1 -817.723,E2 -817.723} C_VEL
LIN {X 0,Y 601.423,Z 369.343,A -85,B 0,C 180,E1 -818.568,E2 -818.568} C_VEL
LIN {X 0,Y 601.455,Z 359.387,A -85,B 0,C 180,E1 -819.415,E2 -819.415} C_VEL
LIN {X 0,Y 601.462,Z 349.574,A -85,B 0,C 180,E1 -820.094,E2 -820.094} C_VEL
LIN {X 0,Y 601.468,Z 338.933,A -85,B 0,C 180,E1 -820.69,E2 -820.69} C_VEL
LIN {X 0,Y 601.519,Z 325.859,A -85,B 0,C 180,E1 -821.253,E2 -821.253} C_VEL
LIN {X 0,Y 601.599,Z 313.051,A -85,B 0,C 180,E1 -821.647,E2 -821.647} C_VEL
LIN {X 0,Y 601.443,Z 302.253,A -85,B 0,C 180,E1 -821.874,E2 -821.874} C_VEL
LIN {X 0,Y 601.342,Z 301.468,A -85,B 0,C 180,E1 -821.908,E2 -821.908} C_VEL
LIN {X 0,Y 601.355,Z 293.664,A -85,B 0,C 180,E1 -824.898,E2 -824.898} C_VEL
LIN {X 0,Y 601.36,Z 286.478,A -85,B 0,C 180,E1 -827.689,E2 -827.689} C_VEL
LIN {X 0,Y 601.377,Z 281.089,A -85,B 0,C 180,E1 -829.81,E2 -829.81} C_VEL
LIN {X 0,Y 601.371,Z 273.903,A -85,B 0,C 180,E1 -832.684,E2 -832.684} C_VEL
LIN {X 0,Y 601.422,Z 266.717,A -85,B 0,C 180,E1 -835.617,E2 -835.617} C_VEL
LIN {X 0,Y 601.357,Z 261.329,A -85,B 0,C 180,E1 -837.87,E2 -837.87} C_VEL
LIN {X 0,Y 601.404,Z 256.065,A -85,B 0,C 180,E1 -840.165,E2 -840.165} C_VEL
LIN {X 0,Y 601.455,Z 250.491,A -85,B 0,C 180,E1 -842.718,E2 -842.718} C_VEL
LIN {X 0,Y 601.479,Z 245.531,A -85,B 0,C 180,E1 -845.121,E2 -845.121} C_VEL
LIN {X 0,Y 601.483,Z 241.007,A -85,B 0,C 180,E1 -847.414,E2 -847.414} C_VEL
LIN {X 0,Y 601.459,Z 236.282,A -85,B 0,C 180,E1 -849.99,E2 -849.99} C_VEL
LIN {X 0,Y 601.459,Z 231.668,A -85,B 0,C 180,E1 -852.665,E2 -852.665} C_VEL
LIN {X 0,Y 601.405,Z 231.071,A -85,B 0,C 180,E1 -853.587,E2 -853.587} C_VEL
LIN {X 0,Y 601.432,Z 231.072,A -85,B 0,C 180,E1 -856.426,E2 -856.426} C_VEL
LIN {X 0,Y 601.404,Z 231.066,A -85,B 0,C 180,E1 -859.426,E2 -859.426} C_VEL
LIN {X 0,Y 601.398,Z 231.07,A -85,B 0,C 180,E1 -861.728,E2 -861.728} C_VEL
LIN {X 0,Y 601.385,Z 231.077,A -85,B 0,C 180,E1 -864.243,E2 -864.243} C_VEL
LIN {X 0,Y 601.419,Z 231.065,A -85,B 0,C 180,E1 -866.684,E2 -866.684} C_VEL
LIN {X 0,Y 601.393,Z 231.067,A -85,B 0,C 180,E1 -869.054,E2 -869.054} C_VEL
LIN {X 0,Y 601.402,Z 231.068,A -85,B 0,C 180,E1 -871.369,E2 -871.369} C_VEL
LIN {X 0,Y 601.409,Z 231.068,A -85,B 0,C 180,E1 -874.379,E2 -874.379} C_VEL
LIN {X 0,Y 601.381,Z 231.069,A -85,B 0,C 180,E1 -876.585,E2 -876.585} C_VEL
LIN {X 0,Y 601.416,Z 231.07,A -85,B 0,C 180,E1 -879.475,E2 -879.475} C_VEL
LIN {X 0,Y 601.376,Z 231.07,A -85,B 0,C 180,E1 -882.308,E2 -882.308} C_VEL
LIN {X 0,Y 601.389,Z 231.068,A -85,B 0,C 180,E1 -884.405,E2 -884.405} C_VEL
LIN {X 0,Y 601.4,Z 231.07,A -85,B 0,C 180,E1 -887.168,E2 -887.168} C_VEL
LIN {X 0,Y 601.415,Z 231.068,A -85,B 0,C 180,E1 -889.901,E2 -889.901} C_VEL
LIN {X 0,Y 601.366,Z 231.071,A -85,B 0,C 180,E1 -892.61,E2 -892.61} C_VEL
LIN {X 0,Y 601.422,Z 231.073,A -85,B 0,C 180,E1 -895.304,E2 -895.304} C_VEL
LIN {X 0,Y 601.393,Z 231.068,A -85,B 0,C 180,E1 -897.987,E2 -897.987} C_VEL
LIN {X 0,Y 601.41,Z 231.065,A -85,B 0,C 180,E1 -899.996,E2 -899.996} C_VEL
LIN {X 0,Y 601.406,Z 231.068,A -85,B 0,C 180,E1 -902.675,E2 -902.675} C_VEL
LIN {X 0,Y 601.426,Z 231.069,A -85,B 0,C 180,E1 -905.36,E2 -905.36} C_VEL
LIN {X 0,Y 601.382,Z 231.068,A -85,B 0,C 180,E1 -908.057,E2 -908.057} C_VEL
LIN {X 0,Y 601.453,Z 231.069,A -85,B 0,C 180,E1 -911.033,E2 -911.033} C_VEL
LIN {X 0,Y 601.376,Z 231.071,A -85,B 0,C 180,E1 -912.349,E2 -912.349} C_VEL
LIN {X 0,Y 600.72,Z 231.161,A -85,B 0,C 180,E1 -912.908,E2 -912.908} C_VEL
LIN {X 0,Y 597.878,Z 231.516,A -85,B 0,C 180,E1 -913.816,E2 -913.816} C_VEL
LIN {X 0,Y 595.466,Z 231.815,A -85,B 0,C 180,E1 -914.546,E2 -914.546} C_VEL
LIN {X 0,Y 594.424,Z 231.942,A -85,B 0,C 180,E1 -915.11,E2 -915.11} C_VEL
LIN {X 0,Y 594.336,Z 231.949,A -85,B 0,C 180,E1 -915.301,E2 -915.301} C_VEL
LIN {X 0,Y 594.317,Z 231.949,A -85,B 0,C 180,E1 -917.901,E2 -917.901} C_VEL
LIN {X 0,Y 594.388,Z 231.949,A -85,B 0,C 180,E1 -920.771,E2 -920.771} C_VEL
LIN {X 0,Y 594.353,Z 231.944,A -85,B 0,C 180,E1 -923.7,E2 -923.7} C_VEL
LIN {X 0,Y 594.354,Z 231.952,A -85,B 0,C 180,E1 -926.695,E2 -926.695} C_VEL
LIN {X 0,Y 594.355,Z 231.947,A -85,B 0,C 180,E1 -928.993,E2 -928.993} C_VEL
LIN {X 0,Y 594.341,Z 231.946,A -85,B 0,C 180,E1 -931.639,E2 -931.639} C_VEL
LIN {X 0,Y 594.36,Z 231.95,A -85,B 0,C 180,E1 -934.574,E2 -934.574} C_VEL
LIN {X 0,Y 594.342,Z 231.946,A -85,B 0,C 180,E1 -937.082,E2 -937.082} C_VEL
LIN {X 0,Y 594.331,Z 231.95,A -85,B 0,C 180,E1 -939.771,E2 -939.771} C_VEL
LIN {X 0,Y 594.356,Z 231.951,A -85,B 0,C 180,E1 -942.368,E2 -942.368} C_VEL
LIN {X 0,Y 594.32,Z 231.948,A -85,B 0,C 180,E1 -945.186,E2 -945.186} C_VEL
LIN {X 0,Y 594.347,Z 231.953,A -85,B 0,C 180,E1 -948.146,E2 -948.146} C_VEL
LIN {X 0,Y 594.337,Z 231.947,A -85,B 0,C 180,E1 -951.192,E2 -951.192} C_VEL
LIN {X 0,Y 594.345,Z 231.953,A -85,B 0,C 180,E1 -953.756,E2 -953.756} C_VEL
LIN {X 0,Y 594.335,Z 231.95,A -85,B 0,C 180,E1 -956.237,E2 -956.237} C_VEL
LIN {X 0,Y 594.334,Z 231.946,A -85,B 0,C 180,E1 -958.648,E2 -958.648} C_VEL
LIN {X 0,Y 594.362,Z 231.944,A -85,B 0,C 180,E1 -961.031,E2 -961.031} C_VEL
LIN {X 0,Y 594.328,Z 231.951,A -85,B 0,C 180,E1 -964.054,E2 -964.054} C_VEL
LIN {X 0,Y 594.344,Z 231.946,A -85,B 0,C 180,E1 -966.295,E2 -966.295} C_VEL
LIN {X 0,Y 594.368,Z 231.947,A -85,B 0,C 180,E1 -969.224,E2 -969.224} C_VEL
LIN {X 0,Y 594.328,Z 231.949,A -85,B 0,C 180,E1 -972.095,E2 -972.095} C_VEL
LIN {X 0,Y 594.319,Z 231.949,A -85,B 0,C 180,E1 -974.218,E2 -974.218} C_VEL
LIN {X 0,Y 594.347,Z 231.95,A -85,B 0,C 180,E1 -977.017,E2 -977.017} C_VEL
LIN {X 0,Y 594.343,Z 231.948,A -85,B 0,C 180,E1 -979.784,E2 -979.784} C_VEL
LIN {X 0,Y 594.354,Z 231.946,A -85,B 0,C 180,E1 -982.527,E2 -982.527} C_VEL
LIN {X 0,Y 594.355,Z 231.952,A -85,B 0,C 180,E1 -985.252,E2 -985.252} C_VEL
LIN {X 0,Y 594.325,Z 231.948,A -85,B 0,C 180,E1 -987.967,E2 -987.967} C_VEL
LIN {X 0,Y 594.378,Z 231.947,A -85,B 0,C 180,E1 -990.677,E2 -990.677} C_VEL
LIN {X 0,Y 594.336,Z 231.95,A -85,B 0,C 180,E1 -993.389,E2 -993.389} C_VEL
LIN {X 0,Y 594.342,Z 231.948,A -85,B 0,C 180,E1 -995.428,E2 -995.428} C_VEL
LIN {X 0,Y 594.354,Z 231.945,A -85,B 0,C 180,E1 -997.473,E2 -997.473} C_VEL
LIN {X 0,Y 594.343,Z 231.948,A -85,B 0,C 180,E1 -1000.216,E2 -1000.216} C_VEL
LIN {X 0,Y 594.347,Z 231.95,A -85,B 0,C 180,E1 -1002.983,E2 -1002.983} C_VEL
LIN {X 0,Y 594.319,Z 231.949,A -85,B 0,C 180,E1 -1005.782,E2 -1005.782} C_VEL
LIN {X 0,Y 594.353,Z 231.953,A -85,B 0,C 180,E1 -1008.618,E2 -1008.618} C_VEL
LIN {X 0,Y 594.318,Z 231.948,A -85,B 0,C 180,E1 -1011.505,E2 -1011.505} C_VEL
LIN {X 0,Y 594.344,Z 231.946,A -85,B 0,C 180,E1 -1013.705,E2 -1013.705} C_VEL
LIN {X 0,Y 594.334,Z 231.951,A -85,B 0,C 180,E1 -1016.701,E2 -1016.701} C_VEL
LIN {X 0,Y 594.36,Z 231.944,A -85,B 0,C 180,E1 -1018.999,E2 -1018.999} C_VEL
LIN {X 0,Y 594.341,Z 231.947,A -85,B 0,C 180,E1 -1021.65,E2 -1021.65} C_VEL
LIN {X 0,Y 594.341,Z 231.949,A -85,B 0,C 180,E1 -1024.582,E2 -1024.582} C_VEL
LIN {X 0,Y 594.329,Z 231.947,A -85,B 0,C 180,E1 -1027.09,E2 -1027.09} C_VEL
LIN {X 0,Y 594.347,Z 231.951,A -85,B 0,C 180,E1 -1029.781,E2 -1029.781} C_VEL
LIN {X 0,Y 594.323,Z 231.951,A -85,B 0,C 180,E1 -1032.378,E2 -1032.378} C_VEL
LIN {X 0,Y 594.334,Z 231.947,A -85,B 0,C 180,E1 -1035.193,E2 -1035.193} C_VEL
LIN {X 0,Y 594.351,Z 231.949,A -85,B 0,C 180,E1 -1038.154,E2 -1038.154} C_VEL
LIN {X 0,Y 594.34,Z 231.948,A -85,B 0,C 180,E1 -1040.325,E2 -1040.325} C_VEL
LIN {X 0,Y 594.342,Z 231.946,A -85,B 0,C 180,E1 -1042.918,E2 -1042.918} C_VEL
LIN {X 0,Y 594.349,Z 231.95,A -85,B 0,C 180,E1 -1045.864,E2 -1045.864} C_VEL
LIN {X 0,Y 594.331,Z 231.947,A -85,B 0,C 180,E1 -1048.654,E2 -1048.654} C_VEL
LIN {X 0,Y 594.358,Z 231.947,A -85,B 0,C 180,E1 -1051.044,E2 -1051.044} C_VEL
LIN {X 0,Y 594.344,Z 231.947,A -85,B 0,C 180,E1 -1053.983,E2 -1053.983} C_VEL
LIN {X 0,Y 594.353,Z 231.944,A -85,B 0,C 180,E1 -1056.3,E2 -1056.3} C_VEL
LIN {X 0,Y 594.388,Z 231.949,A -85,B 0,C 180,E1 -1059.229,E2 -1059.229} C_VEL
LIN {X 0,Y 594.316,Z 231.949,A -85,B 0,C 180,E1 -1062.099,E2 -1062.099} C_VEL
LIN {X 0,Y 594.337,Z 231.946,A -85,B 0,C 180,E1 -1064.223,E2 -1064.223} C_VEL
LIN {X 0,Y 594.344,Z 231.954,A -85,B 0,C 180,E1 -1067.021,E2 -1067.021} C_VEL
LIN {X 0,Y 594.382,Z 231.95,A -85,B 0,C 180,E1 -1069.1,E2 -1069.1} C_VEL
LIN {X 0,Y 594.336,Z 231.946,A -85,B 0,C 180,E1 -1071.847,E2 -1071.847} C_VEL
LIN {X 0,Y 594.385,Z 231.945,A -85,B 0,C 180,E1 -1074.576,E2 -1074.576} C_VEL
LIN {X 0,Y 594.376,Z 231.944,A -85,B 0,C 180,E1 -1077.293,E2 -1077.293} C_VEL
LIN {X 0,Y 594.381,Z 231.941,A -85,B 0,C 180,E1 -1080.004,E2 -1080.004} C_VEL
LIN {X 0,Y 594.402,Z 231.948,A -85,B 0,C 180,E1 -1082.715,E2 -1082.715} C_VEL
LIN {X 0,Y 594.356,Z 231.944,A -85,B 0,C 180,E1 -1085.432,E2 -1085.432} C_VEL
LIN {X 0,Y 594.337,Z 231.946,A -85,B 0,C 180,E1 -1087.477,E2 -1087.477} C_VEL
LIN {X 0,Y 594.374,Z 231.947,A -85,B 0,C 180,E1 -1090.22,E2 -1090.22} C_VEL
LIN {X 0,Y 594.346,Z 231.947,A -85,B 0,C 180,E1 -1092.987,E2 -1092.987} C_VEL
LIN {X 0,Y 594.355,Z 231.945,A -85,B 0,C 180,E1 -1095.082,E2 -1095.082} C_VEL
LIN {X 0,Y 594.365,Z 231.943,A -85,B 0,C 180,E1 -1097.197,E2 -1097.197} C_VEL
LIN {X 0,Y 594.36,Z 231.95,A -85,B 0,C 180,E1 -1100.057,E2 -1100.057} C_VEL
LIN {X 0,Y 594.35,Z 231.945,A -85,B 0,C 180,E1 -1102.971,E2 -1102.971} C_VEL
LIN {X 0,Y 594.356,Z 231.944,A -85,B 0,C 180,E1 -1105.197,E2 -1105.197} C_VEL
LIN {X 0,Y 594.358,Z 231.951,A -85,B 0,C 180,E1 -1108.231,E2 -1108.231} C_VEL
LIN {X 0,Y 594.364,Z 231.945,A -85,B 0,C 180,E1 -1110.563,E2 -1110.563} C_VEL
LIN {X 0,Y 594.373,Z 231.941,A -85,B 0,C 180,E1 -1112.953,E2 -1112.953} C_VEL
LIN {X 0,Y 594.325,Z 231.95,A -85,B 0,C 180,E1 -1115.413,E2 -1115.413} C_VEL
LIN {X 0,Y 594.373,Z 231.95,A -85,B 0,C 180,E1 -1117.944,E2 -1117.944} C_VEL
LIN {X 0,Y 594.369,Z 231.943,A -85,B 0,C 180,E1 -1120.823,E2 -1120.823} C_VEL
LIN {X 0,Y 594.363,Z 231.952,A -85,B 0,C 180,E1 -1123.84,E2 -1123.84} C_VEL
LIN {X 0,Y 594.363,Z 231.954,A -85,B 0,C 180,E1 -1126.702,E2 -1126.702} C_VEL
LIN {X 0,Y 594.481,Z 234.934,A -85,B 0,C 180,E1 -1128.546,E2 -1128.546} C_VEL
LIN {X 0,Y 594.513,Z 239.76,A -85,B 0,C 180,E1 -1131.282,E2 -1131.282} C_VEL
LIN {X 0,Y 594.47,Z 244.432,A -85,B 0,C 180,E1 -1133.765,E2 -1133.765} C_VEL
LIN {X 0,Y 594.447,Z 249.389,A -85,B 0,C 180,E1 -1136.244,E2 -1136.244} C_VEL
LIN {X 0,Y 594.399,Z 254.436,A -85,B 0,C 180,E1 -1138.652,E2 -1138.652} C_VEL
LIN {X 0,Y 594.338,Z 259.709,A -85,B 0,C 180,E1 -1141.052,E2 -1141.052} C_VEL
LIN {X 0,Y 594.333,Z 264.925,A -85,B 0,C 180,E1 -1143.299,E2 -1143.299} C_VEL
LIN {X 0,Y 594.335,Z 270.376,A -85,B 0,C 180,E1 -1145.58,E2 -1145.58} C_VEL
LIN {X 0,Y 594.29,Z 277.496,A -85,B 0,C 180,E1 -1148.494,E2 -1148.494} C_VEL
LIN {X 0,Y 594.305,Z 284.682,A -85,B 0,C 180,E1 -1151.38,E2 -1151.38} C_VEL
LIN {X 0,Y 594.258,Z 291.868,A -85,B 0,C 180,E1 -1154.217,E2 -1154.217} C_VEL
LIN {X 0,Y 594.254,Z 297.257,A -85,B 0,C 180,E1 -1156.318,E2 -1156.318} C_VEL
LIN {X 0,Y 594.271,Z 301.532,A -85,B 0,C 180,E1 -1157.969,E2 -1157.969} C_VEL
LIN {X 0,Y 594.67,Z 307.54,A -85,B 0,C 180,E1 -1158.086,E2 -1158.086} C_VEL
LIN {X 0,Y 594.601,Z 319.844,A -85,B 0,C 180,E1 -1158.409,E2 -1158.409} C_VEL
LIN {X 0,Y 594.531,Z 331.968,A -85,B 0,C 180,E1 -1158.86,E2 -1158.86} C_VEL
LIN {X 0,Y 594.479,Z 343.774,A -85,B 0,C 180,E1 -1159.442,E2 -1159.442} C_VEL
LIN {X 0,Y 594.449,Z 354.751,A -85,B 0,C 180,E1 -1160.129,E2 -1160.129} C_VEL
LIN {X 0,Y 594.404,Z 365.587,A -85,B 0,C 180,E1 -1160.987,E2 -1160.987} C_VEL
LIN {X 0,Y 594.366,Z 374.396,A -85,B 0,C 180,E1 -1161.843,E2 -1161.843} C_VEL
LIN {X 0,Y 594.306,Z 383.006,A -85,B 0,C 180,E1 -1162.867,E2 -1162.867} C_VEL
LIN {X 0,Y 594.289,Z 389.871,A -85,B 0,C 180,E1 -1163.89,E2 -1163.89} C_VEL
LIN {X 0,Y 594.254,Z 395.365,A -85,B 0,C 180,E1 -1164.911,E2 -1164.911} C_VEL
LIN {X 0,Y 594.263,Z 399.669,A -85,B 0,C 180,E1 -1165.931,E2 -1165.931} C_VEL
LIN {X 0,Y 594.267,Z 401.962,A -85,B 0,C 180,E1 -1166.61,E2 -1166.61} C_VEL
LIN {X 0,Y 594.226,Z 403.8,A -85,B 0,C 180,E1 -1167.288,E2 -1167.288} C_VEL
LIN {X 0,Y 594.242,Z 405.193,A -85,B 0,C 180,E1 -1167.967,E2 -1167.967} C_VEL
LIN {X 0,Y 594.247,Z 406.187,A -85,B 0,C 180,E1 -1168.645,E2 -1168.645} C_VEL
LIN {X 0,Y 594.239,Z 406.782,A -85,B 0,C 180,E1 -1169.322,E2 -1169.322} C_VEL
LIN {X 0,Y 594.236,Z 406.983,A -85,B 0,C 180,E1 -1170,E2 -1170} C_VEL
LIN {X 0,Y 594.239,Z 406.782,A -85,B 0,C 180,E1 -1170.678,E2 -1170.678} C_VEL
LIN {X 0,Y 594.247,Z 406.187,A -85,B 0,C 180,E1 -1171.355,E2 -1171.355} C_VEL
LIN {X 0,Y 594.242,Z 405.193,A -85,B 0,C 180,E1 -1172.033,E2 -1172.033} C_VEL
LIN {X 0,Y 594.226,Z 403.8,A -85,B 0,C 180,E1 -1172.712,E2 -1172.712} C_VEL
LIN {X 0,Y 594.289,Z 400.89,A -85,B 0,C 180,E1 -1173.729,E2 -1173.729} C_VEL
LIN {X 0,Y 594.241,Z 396.942,A -85,B 0,C 180,E1 -1174.749,E2 -1174.749} C_VEL
LIN {X 0,Y 594.3,Z 391.848,A -85,B 0,C 180,E1 -1175.769,E2 -1175.769} C_VEL
LIN {X 0,Y 594.317,Z 385.464,A -85,B 0,C 180,E1 -1176.791,E2 -1176.791} C_VEL
LIN {X 0,Y 594.347,Z 377.487,A -85,B 0,C 180,E1 -1177.815,E2 -1177.815} C_VEL
LIN {X 0,Y 594.378,Z 369.346,A -85,B 0,C 180,E1 -1178.671,E2 -1178.671} C_VEL
LIN {X 0,Y 594.418,Z 359.374,A -85,B 0,C 180,E1 -1179.528,E2 -1179.528} C_VEL
LIN {X 0,Y 594.452,Z 349.558,A -85,B 0,C 180,E1 -1180.215,E2 -1180.215} C_VEL
LIN {X 0,Y 594.484,Z 338.938,A -85,B 0,C 180,E1 -1180.817,E2 -1180.817} C_VEL
LIN {X 0,Y 594.549,Z 326.202,A -85,B 0,C 180,E1 -1181.374,E2 -1181.374} C_VEL
LIN {X 0,Y 594.656,Z 313.892,A -85,B 0,C 180,E1 -1181.763,E2 -1181.763} C_VEL
LIN {X 0,Y 594.533,Z 303.29,A -85,B 0,C 180,E1 -1181.997,E2 -1181.997} C_VEL
LIN {X 0,Y 594.275,Z 301.468,A -85,B 0,C 180,E1 -1182.052,E2 -1182.052} C_VEL
LIN {X 0,Y 594.272,Z 293.664,A -85,B 0,C 180,E1 -1185.08,E2 -1185.08} C_VEL
LIN {X 0,Y 594.291,Z 288.275,A -85,B 0,C 180,E1 -1187.196,E2 -1187.196} C_VEL
LIN {X 0,Y 594.292,Z 282.885,A -85,B 0,C 180,E1 -1189.336,E2 -1189.336} C_VEL
LIN {X 0,Y 594.314,Z 275.699,A -85,B 0,C 180,E1 -1192.235,E2 -1192.235} C_VEL
LIN {X 0,Y 594.336,Z 268.514,A -85,B 0,C 180,E1 -1195.194,E2 -1195.194} C_VEL
LIN {X 0,Y 594.346,Z 263.016,A -85,B 0,C 180,E1 -1197.517,E2 -1197.517} C_VEL
LIN {X 0,Y 594.372,Z 256.672,A -85,B 0,C 180,E1 -1200.324,E2 -1200.324} C_VEL
LIN {X 0,Y 594.428,Z 251.059,A -85,B 0,C 180,E1 -1202.946,E2 -1202.946} C_VEL
LIN {X 0,Y 594.457,Z 246.079,A -85,B 0,C 180,E1 -1205.401,E2 -1205.401} C_VEL
LIN {X 0,Y 594.483,Z 241.2,A -85,B 0,C 180,E1 -1207.932,E2 -1207.932} C_VEL
LIN {X 0,Y 594.504,Z 236.012,A -85,B 0,C 180,E1 -1210.834,E2 -1210.834} C_VEL
LIN {X 0,Y 594.432,Z 232.643,A -85,B 0,C 180,E1 -1212.857,E2 -1212.857} C_VEL
LIN {X 0,Y 594.363,Z 231.953,A -85,B 0,C 180,E1 -1213.298,E2 -1213.298} C_VEL
LIN {X 0,Y 594.363,Z 231.952,A -85,B 0,C 180,E1 -1216.16,E2 -1216.16} C_VEL
LIN {X 0,Y 594.369,Z 231.943,A -85,B 0,C 180,E1 -1219.177,E2 -1219.177} C_VEL
LIN {X 0,Y 594.373,Z 231.95,A -85,B 0,C 180,E1 -1222.056,E2 -1222.056} C_VEL
LIN {X 0,Y 594.325,Z 231.95,A -85,B 0,C 180,E1 -1224.678,E2 -1224.678} C_VEL
LIN {X 0,Y 594.373,Z 231.942,A -85,B 0,C 180,E1 -1227.087,E2 -1227.087} C_VEL
LIN {X 0,Y 594.369,Z 231.947,A -85,B 0,C 180,E1 -1229.672,E2 -1229.672} C_VEL
LIN {X 0,Y 594.342,Z 231.947,A -85,B 0,C 180,E1 -1232.479,E2 -1232.479} C_VEL
LIN {X 0,Y 594.356,Z 231.944,A -85,B 0,C 180,E1 -1234.803,E2 -1234.803} C_VEL
LIN {X 0,Y 594.356,Z 231.946,A -85,B 0,C 180,E1 -1237.264,E2 -1237.264} C_VEL
LIN {X 0,Y 594.36,Z 231.95,A -85,B 0,C 180,E1 -1239.943,E2 -1239.943} C_VEL
LIN {X 0,Y 594.365,Z 231.943,A -85,B 0,C 180,E1 -1242.803,E2 -1242.803} C_VEL
LIN {X 0,Y 594.383,Z 231.946,A -85,B 0,C 180,E1 -1245.824,E2 -1245.824} C_VEL
LIN {X 0,Y 594.365,Z 231.943,A -85,B 0,C 180,E1 -1248.4,E2 -1248.4} C_VEL
LIN {X 0,Y 594.369,Z 231.947,A -85,B 0,C 180,E1 -1251.154,E2 -1251.154} C_VEL
LIN {X 0,Y 594.342,Z 231.948,A -85,B 0,C 180,E1 -1253.887,E2 -1253.887} C_VEL
LIN {X 0,Y 594.332,Z 231.948,A -85,B 0,C 180,E1 -1255.928,E2 -1255.928} C_VEL
LIN {X 0,Y 594.366,Z 231.943,A -85,B 0,C 180,E1 -1257.963,E2 -1257.963} C_VEL
LIN {X 0,Y 594.381,Z 231.941,A -85,B 0,C 180,E1 -1259.996,E2 -1259.996} C_VEL
LIN {X 0,Y 594.376,Z 231.944,A -85,B 0,C 180,E1 -1262.707,E2 -1262.707} C_VEL
LIN {X 0,Y 594.385,Z 231.945,A -85,B 0,C 180,E1 -1265.424,E2 -1265.424} C_VEL
LIN {X 0,Y 594.336,Z 231.946,A -85,B 0,C 180,E1 -1268.153,E2 -1268.153} C_VEL
LIN {X 0,Y 594.425,Z 231.943,A -85,B 0,C 180,E1 -1271.098,E2 -1271.098} C_VEL
LIN {X 0,Y 594.362,Z 231.945,A -85,B 0,C 180,E1 -1274.373,E2 -1274.373} C_VEL
LIN {X 0,Y 594.336,Z 231.949,A -85,B 0,C 180,E1 -1275.301,E2 -1275.301} C_VEL
LIN {X 0,Y 593.655,Z 232.033,A -85,B 0,C 180,E1 -1275.867,E2 -1275.867} C_VEL
LIN {X 0,Y 590.782,Z 232.399,A -85,B 0,C 180,E1 -1276.785,E2 -1276.785} C_VEL
LIN {X 0,Y 588.372,Z 232.694,A -85,B 0,C 180,E1 -1277.523,E2 -1277.523} C_VEL
LIN {X 0,Y 587.352,Z 232.817,A -85,B 0,C 180,E1 -1278.093,E2 -1278.093} C_VEL
LIN {X 0,Y 587.277,Z 232.827,A -85,B 0,C 180,E1 -1278.286,E2 -1278.286} C_VEL
LIN {X 0,Y 587.329,Z 232.824,A -85,B 0,C 180,E1 -1281.04,E2 -1281.04} C_VEL
LIN {X 0,Y 587.301,Z 232.824,A -85,B 0,C 180,E1 -1284.002,E2 -1284.002} C_VEL
LIN {X 0,Y 587.303,Z 232.827,A -85,B 0,C 180,E1 -1286.274,E2 -1286.274} C_VEL
LIN {X 0,Y 587.319,Z 232.822,A -85,B 0,C 180,E1 -1289.13,E2 -1289.13} C_VEL
LIN {X 0,Y 587.312,Z 232.823,A -85,B 0,C 180,E1 -1291.833,E2 -1291.833} C_VEL
LIN {X 0,Y 587.319,Z 232.83,A -85,B 0,C 180,E1 -1294.346,E2 -1294.346} C_VEL
LIN {X 0,Y 587.309,Z 232.825,A -85,B 0,C 180,E1 -1296.742,E2 -1296.742} C_VEL
LIN {X 0,Y 587.295,Z 232.823,A -85,B 0,C 180,E1 -1299.355,E2 -1299.355} C_VEL
LIN {X 0,Y 587.317,Z 232.829,A -85,B 0,C 180,E1 -1302.107,E2 -1302.107} C_VEL
LIN {X 0,Y 587.276,Z 232.826,A -85,B 0,C 180,E1 -1305.086,E2 -1305.086} C_VEL
LIN {X 0,Y 587.297,Z 232.831,A -85,B 0,C 180,E1 -1307.924,E2 -1307.924} C_VEL
LIN {X 0,Y 587.304,Z 232.823,A -85,B 0,C 180,E1 -1310.639,E2 -1310.639} C_VEL
LIN {X 0,Y 587.296,Z 232.825,A -85,B 0,C 180,E1 -1313.288,E2 -1313.288} C_VEL
LIN {X 0,Y 587.319,Z 232.829,A -85,B 0,C 180,E1 -1315.778,E2 -1315.778} C_VEL
LIN {X 0,Y 587.304,Z 232.825,A -85,B 0,C 180,E1 -1318.23,E2 -1318.23} C_VEL
LIN {X 0,Y 587.318,Z 232.82,A -85,B 0,C 180,E1 -1320.858,E2 -1320.858} C_VEL
LIN {X 0,Y 587.304,Z 232.83,A -85,B 0,C 180,E1 -1323.814,E2 -1323.814} C_VEL
LIN {X 0,Y 587.317,Z 232.821,A -85,B 0,C 180,E1 -1326.742,E2 -1326.742} C_VEL
LIN {X 0,Y 587.289,Z 232.831,A -85,B 0,C 180,E1 -1329.694,E2 -1329.694} C_VEL
LIN {X 0,Y 587.282,Z 232.829,A -85,B 0,C 180,E1 -1331.872,E2 -1331.872} C_VEL
LIN {X 0,Y 587.282,Z 232.827,A -85,B 0,C 180,E1 -1334.024,E2 -1334.024} C_VEL
LIN {X 0,Y 587.288,Z 232.828,A -85,B 0,C 180,E1 -1336.858,E2 -1336.858} C_VEL
LIN {X 0,Y 587.294,Z 232.828,A -85,B 0,C 180,E1 -1339.66,E2 -1339.66} C_VEL
LIN {X 0,Y 587.317,Z 232.822,A -85,B 0,C 180,E1 -1342.436,E2 -1342.436} C_VEL
LIN {X 0,Y 587.323,Z 232.829,A -85,B 0,C 180,E1 -1345.195,E2 -1345.195} C_VEL
LIN {X 0,Y 587.296,Z 232.824,A -85,B 0,C 180,E1 -1347.943,E2 -1347.943} C_VEL
LIN {X 0,Y 587.346,Z 232.823,A -85,B 0,C 180,E1 -1350.686,E2 -1350.686} C_VEL
LIN {X 0,Y 587.286,Z 232.827,A -85,B 0,C 180,E1 -1353.43,E2 -1353.43} C_VEL
LIN {X 0,Y 587.305,Z 232.824,A -85,B 0,C 180,E1 -1355.493,E2 -1355.493} C_VEL
LIN {X 0,Y 587.318,Z 232.822,A -85,B 0,C 180,E1 -1357.564,E2 -1357.564} C_VEL
LIN {X 0,Y 587.294,Z 232.828,A -85,B 0,C 180,E1 -1360.34,E2 -1360.34} C_VEL
LIN {X 0,Y 587.288,Z 232.828,A -85,B 0,C 180,E1 -1363.142,E2 -1363.142} C_VEL
LIN {X 0,Y 587.282,Z 232.827,A -85,B 0,C 180,E1 -1365.976,E2 -1365.976} C_VEL
LIN {X 0,Y 587.314,Z 232.826,A -85,B 0,C 180,E1 -1368.849,E2 -1368.849} C_VEL
LIN {X 0,Y 587.28,Z 232.826,A -85,B 0,C 180,E1 -1371.775,E2 -1371.775} C_VEL
LIN {X 0,Y 587.314,Z 232.828,A -85,B 0,C 180,E1 -1374.589,E2 -1374.589} C_VEL
LIN {X 0,Y 587.279,Z 232.826,A -85,B 0,C 180,E1 -1377.048,E2 -1377.048} C_VEL
LIN {X 0,Y 587.315,Z 232.821,A -85,B 0,C 180,E1 -1379.38,E2 -1379.38} C_VEL
LIN {X 0,Y 587.306,Z 232.826,A -85,B 0,C 180,E1 -1381.843,E2 -1381.843} C_VEL
LIN {X 0,Y 587.306,Z 232.829,A -85,B 0,C 180,E1 -1384.354,E2 -1384.354} C_VEL
LIN {X 0,Y 587.295,Z 232.824,A -85,B 0,C 180,E1 -1386.75,E2 -1386.75} C_VEL
LIN {X 0,Y 587.304,Z 232.823,A -85,B 0,C 180,E1 -1389.361,E2 -1389.361} C_VEL
LIN {X 0,Y 587.312,Z 232.829,A -85,B 0,C 180,E1 -1392.115,E2 -1392.115} C_VEL
LIN {X 0,Y 587.283,Z 232.825,A -85,B 0,C 180,E1 -1395.095,E2 -1395.095} C_VEL
LIN {X 0,Y 587.303,Z 232.83,A -85,B 0,C 180,E1 -1397.932,E2 -1397.932} C_VEL
LIN {X 0,Y 587.295,Z 232.823,A -85,B 0,C 180,E1 -1400.645,E2 -1400.645} C_VEL
LIN {X 0,Y 587.31,Z 232.825,A -85,B 0,C 180,E1 -1403.296,E2 -1403.296} C_VEL
LIN {X 0,Y 587.331,Z 232.826,A -85,B 0,C 180,E1 -1405.785,E2 -1405.785} C_VEL
LIN {X 0,Y 587.309,Z 232.822,A -85,B 0,C 180,E1 -1408.236,E2 -1408.236} C_VEL
LIN {X 0,Y 587.319,Z 232.822,A -85,B 0,C 180,E1 -1410.87,E2 -1410.87} C_VEL
LIN {X 0,Y 587.321,Z 232.824,A -85,B 0,C 180,E1 -1413.824,E2 -1413.824} C_VEL
LIN {X 0,Y 587.301,Z 232.824,A -85,B 0,C 180,E1 -1415.998,E2 -1415.998} C_VEL
LIN {X 0,Y 587.319,Z 232.825,A -85,B 0,C 180,E1 -1418.968,E2 -1418.968} C_VEL
LIN {X 0,Y 587.325,Z 232.829,A -85,B 0,C 180,E1 -1421.156,E2 -1421.156} C_VEL
LIN {X 0,Y 587.294,Z 232.824,A -85,B 0,C 180,E1 -1424.029,E2 -1424.029} C_VEL
LIN {X 0,Y 587.326,Z 232.819,A -85,B 0,C 180,E1 -1426.158,E2 -1426.158} C_VEL
LIN {X 0,Y 587.373,Z 232.823,A -85,B 0,C 180,E1 -1428.968,E2 -1428.968} C_VEL
LIN {X 0,Y 587.303,Z 232.823,A -85,B 0,C 180,E1 -1431.748,E2 -1431.748} C_VEL
LIN {X 0,Y 587.345,Z 232.821,A -85,B 0,C 180,E1 -1434.511,E2 -1434.511} C_VEL
LIN {X 0,Y 587.345,Z 232.82,A -85,B 0,C 180,E1 -1437.261,E2 -1437.261} C_VEL
LIN {X 0,Y 587.352,Z 232.817,A -85,B 0,C 180,E1 -1440.004,E2 -1440.004} C_VEL
LIN {X 0,Y 587.364,Z 232.824,A -85,B 0,C 180,E1 -1442.747,E2 -1442.747} C_VEL
LIN {X 0,Y 587.323,Z 232.82,A -85,B 0,C 180,E1 -1445.497,E2 -1445.497} C_VEL
LIN {X 0,Y 587.299,Z 232.823,A -85,B 0,C 180,E1 -1447.568,E2 -1447.568} C_VEL
LIN {X 0,Y 587.323,Z 232.827,A -85,B 0,C 180,E1 -1450.344,E2 -1450.344} C_VEL
LIN {X 0,Y 587.297,Z 232.824,A -85,B 0,C 180,E1 -1453.145,E2 -1453.145} C_VEL
LIN {X 0,Y 587.313,Z 232.821,A -85,B 0,C 180,E1 -1455.267,E2 -1455.267} C_VEL
LIN {X 0,Y 587.301,Z 232.822,A -85,B 0,C 180,E1 -1457.411,E2 -1457.411} C_VEL
LIN {X 0,Y 587.301,Z 232.823,A -85,B 0,C 180,E1 -1459.579,E2 -1459.579} C_VEL
LIN {X 0,Y 587.31,Z 232.825,A -85,B 0,C 180,E1 -1461.778,E2 -1461.778} C_VEL
LIN {X 0,Y 587.345,Z 232.819,A -85,B 0,C 180,E1 -1464.762,E2 -1464.762} C_VEL
LIN {X 0,Y 587.3,Z 232.829,A -85,B 0,C 180,E1 -1467.823,E2 -1467.823} C_VEL
LIN {X 0,Y 587.32,Z 232.823,A -85,B 0,C 180,E1 -1470.509,E2 -1470.509} C_VEL
LIN {X 0,Y 587.336,Z 232.818,A -85,B 0,C 180,E1 -1473.113,E2 -1473.113} C_VEL
LIN {X 0,Y 587.276,Z 232.83,A -85,B 0,C 180,E1 -1475.537,E2 -1475.537} C_VEL
LIN {X 0,Y 587.331,Z 232.829,A -85,B 0,C 180,E1 -1477.839,E2 -1477.839} C_VEL
LIN {X 0,Y 587.305,Z 232.826,A -85,B 0,C 180,E1 -1480.257,E2 -1480.257} C_VEL
LIN {X 0,Y 587.299,Z 232.826,A -85,B 0,C 180,E1 -1483.118,E2 -1483.118} C_VEL
LIN {X 0,Y 587.3,Z 232.832,A -85,B 0,C 180,E1 -1486.049,E2 -1486.049} C_VEL
LIN {X 0,Y 587.436,Z 233.701,A -85,B 0,C 180,E1 -1487.006,E2 -1487.006} C_VEL
LIN {X 0,Y 587.493,Z 236.794,A -85,B 0,C 180,E1 -1488.91,E2 -1488.91} C_VEL
LIN {X 0,Y 587.484,Z 241.412,A -85,B 0,C 180,E1 -1491.534,E2 -1491.534} C_VEL
LIN {X 0,Y 587.445,Z 246.209,A -85,B 0,C 180,E1 -1494.112,E2 -1494.112} C_VEL
LIN {X 0,Y 587.403,Z 251.74,A -85,B 0,C 180,E1 -1496.881,E2 -1496.881} C_VEL
LIN {X 0,Y 587.322,Z 257.963,A -85,B 0,C 180,E1 -1499.83,E2 -1499.83} C_VEL
LIN {X 0,Y 587.298,Z 263.503,A -85,B 0,C 180,E1 -1502.319,E2 -1502.319} C_VEL
LIN {X 0,Y 587.268,Z 268.523,A -85,B 0,C 180,E1 -1504.481,E2 -1504.481} C_VEL
LIN {X 0,Y 587.258,Z 275.7,A -85,B 0,C 180,E1 -1507.483,E2 -1507.483} C_VEL
LIN {X 0,Y 587.207,Z 281.089,A -85,B 0,C 180,E1 -1509.691,E2 -1509.691} C_VEL
LIN {X 0,Y 587.198,Z 286.478,A -85,B 0,C 180,E1 -1511.87,E2 -1511.87} C_VEL
LIN {X 0,Y 587.19,Z 291.868,A -85,B 0,C 180,E1 -1514.021,E2 -1514.021} C_VEL
LIN {X 0,Y 587.19,Z 297.257,A -85,B 0,C 180,E1 -1516.151,E2 -1516.151} C_VEL
LIN {X 0,Y 587.152,Z 301.524,A -85,B 0,C 180,E1 -1517.821,E2 -1517.821} C_VEL
LIN {X 0,Y 587.726,Z 306.418,A -85,B 0,C 180,E1 -1517.921,E2 -1517.921} C_VEL
LIN {X 0,Y 587.654,Z 319.828,A -85,B 0,C 180,E1 -1518.27,E2 -1518.27} C_VEL
LIN {X 0,Y 587.55,Z 331.682,A -85,B 0,C 180,E1 -1518.714,E2 -1518.714} C_VEL
LIN {X 0,Y 587.497,Z 343.774,A -85,B 0,C 180,E1 -1519.315,E2 -1519.315} C_VEL
LIN {X 0,Y 587.449,Z 354.751,A -85,B 0,C 180,E1 -1520.01,E2 -1520.01} C_VEL
LIN {X 0,Y 587.385,Z 363.642,A -85,B 0,C 180,E1 -1520.705,E2 -1520.705} C_VEL
LIN {X 0,Y 587.331,Z 372.764,A -85,B 0,C 180,E1 -1521.571,E2 -1521.571} C_VEL
LIN {X 0,Y 587.272,Z 380.312,A -85,B 0,C 180,E1 -1522.436,E2 -1522.436} C_VEL
LIN {X 0,Y 587.214,Z 387.303,A -85,B 0,C 180,E1 -1523.405,E2 -1523.405} C_VEL
LIN {X 0,Y 587.211,Z 393.682,A -85,B 0,C 180,E1 -1524.506,E2 -1524.506} C_VEL
LIN {X 0,Y 587.189,Z 398.378,A -85,B 0,C 180,E1 -1525.538,E2 -1525.538} C_VEL
LIN {X 0,Y 587.194,Z 401.964,A -85,B 0,C 180,E1 -1526.569,E2 -1526.569} C_VEL
LIN {X 0,Y 587.132,Z 403.795,A -85,B 0,C 180,E1 -1527.256,E2 -1527.256} C_VEL
LIN {X 0,Y 587.147,Z 406.189,A -85,B 0,C 180,E1 -1528.628,E2 -1528.628} C_VEL
LIN {X 0,Y 587.14,Z 406.782,A -85,B 0,C 180,E1 -1529.314,E2 -1529.314} C_VEL
LIN {X 0,Y 587.14,Z 406.782,A -85,B 0,C 180,E1 -1530.686,E2 -1530.686} C_VEL
LIN {X 0,Y 587.147,Z 406.189,A -85,B 0,C 180,E1 -1531.372,E2 -1531.372} C_VEL
LIN {X 0,Y 587.132,Z 403.795,A -85,B 0,C 180,E1 -1532.744,E2 -1532.744} C_VEL
LIN {X 0,Y 587.213,Z 400.883,A -85,B 0,C 180,E1 -1533.774,E2 -1533.774} C_VEL
LIN {X 0,Y 587.146,Z 396.934,A -85,B 0,C 180,E1 -1534.806,E2 -1534.806} C_VEL
LIN {X 0,Y 587.23,Z 391.839,A -85,B 0,C 180,E1 -1535.839,E2 -1535.839} C_VEL
LIN {X 0,Y 587.231,Z 385.455,A -85,B 0,C 180,E1 -1536.873,E2 -1536.873} C_VEL
LIN {X 0,Y 587.288,Z 377.49,A -85,B 0,C 180,E1 -1537.91,E2 -1537.91} C_VEL
LIN {X 0,Y 587.336,Z 369.349,A -85,B 0,C 180,E1 -1538.775,E2 -1538.775} C_VEL
LIN {X 0,Y 587.389,Z 359.362,A -85,B 0,C 180,E1 -1539.643,E2 -1539.643} C_VEL
LIN {X 0,Y 587.441,Z 349.543,A -85,B 0,C 180,E1 -1540.338,E2 -1540.338} C_VEL
LIN {X 0,Y 587.495,Z 338.939,A -85,B 0,C 180,E1 -1540.947,E2 -1540.947} C_VEL
LIN {X 0,Y 587.594,Z 325.424,A -85,B 0,C 180,E1 -1541.541,E2 -1541.541} C_VEL
LIN {X 0,Y 587.71,Z 312.987,A -85,B 0,C 180,E1 -1541.926,E2 -1541.926} C_VEL
LIN {X 0,Y 587.566,Z 304.126,A -85,B 0,C 180,E1 -1542.126,E2 -1542.126} C_VEL
LIN {X 0,Y 587.152,Z 301.524,A -85,B 0,C 180,E1 -1542.179,E2 -1542.179} C_VEL
LIN {X 0,Y 587.206,Z 295.461,A -85,B 0,C 180,E1 -1544.556,E2 -1544.556} C_VEL
LIN {X 0,Y 587.214,Z 288.275,A -85,B 0,C 180,E1 -1547.41,E2 -1547.41} C_VEL
LIN {X 0,Y 587.217,Z 282.885,A -85,B 0,C 180,E1 -1549.579,E2 -1549.579} C_VEL
LIN {X 0,Y 587.246,Z 277.496,A -85,B 0,C 180,E1 -1551.777,E2 -1551.777} C_VEL
LIN {X 0,Y 587.255,Z 270.31,A -85,B 0,C 180,E1 -1554.762,E2 -1554.762} C_VEL
LIN {X 0,Y 587.289,Z 264.964,A -85,B 0,C 180,E1 -1557.048,E2 -1557.048} C_VEL
LIN {X 0,Y 587.299,Z 259.668,A -85,B 0,C 180,E1 -1559.381,E2 -1559.381} C_VEL
LIN {X 0,Y 587.367,Z 254.408,A -85,B 0,C 180,E1 -1561.837,E2 -1561.837} C_VEL
LIN {X 0,Y 587.44,Z 249.201,A -85,B 0,C 180,E1 -1564.359,E2 -1564.359} C_VEL
LIN {X 0,Y 587.493,Z 244.606,A -85,B 0,C 180,E1 -1566.735,E2 -1566.735} C_VEL
LIN {X 0,Y 587.496,Z 239.799,A -85,B 0,C 180,E1 -1569.346,E2 -1569.346} C_VEL
LIN {X 0,Y 587.519,Z 235.074,A -85,B 0,C 180,E1 -1572.125,E2 -1572.125} C_VEL
LIN {X 0,Y 587.401,Z 233.5,A -85,B 0,C 180,E1 -1573.125,E2 -1573.125} C_VEL
LIN {X 0,Y 587.305,Z 232.832,A -85,B 0,C 180,E1 -1574.109,E2 -1574.109} C_VEL
LIN {X 0,Y 587.293,Z 232.826,A -85,B 0,C 180,E1 -1576.989,E2 -1576.989} C_VEL
LIN {X 0,Y 587.305,Z 232.826,A -85,B 0,C 180,E1 -1579.743,E2 -1579.743} C_VEL
LIN {X 0,Y 587.339,Z 232.825,A -85,B 0,C 180,E1 -1582.39,E2 -1582.39} C_VEL
LIN {X 0,Y 587.349,Z 232.822,A -85,B 0,C 180,E1 -1585.777,E2 -1585.777} C_VEL
LIN {X 0,Y 587.332,Z 232.825,A -85,B 0,C 180,E1 -1588.228,E2 -1588.228} C_VEL
LIN {X 0,Y 587.342,Z 232.817,A -85,B 0,C 180,E1 -1590.866,E2 -1590.866} C_VEL
LIN {X 0,Y 587.307,Z 232.831,A -85,B 0,C 180,E1 -1593.827,E2 -1593.827} C_VEL
LIN {X 0,Y 587.325,Z 232.827,A -85,B 0,C 180,E1 -1595.99,E2 -1595.99} C_VEL
LIN {X 0,Y 587.31,Z 232.825,A -85,B 0,C 180,E1 -1598.222,E2 -1598.222} C_VEL
LIN {X 0,Y 587.329,Z 232.821,A -85,B 0,C 180,E1 -1601.148,E2 -1601.148} C_VEL
LIN {X 0,Y 587.302,Z 232.826,A -85,B 0,C 180,E1 -1604.021,E2 -1604.021} C_VEL
LIN {X 0,Y 587.345,Z 232.819,A -85,B 0,C 180,E1 -1606.151,E2 -1606.151} C_VEL
LIN {X 0,Y 587.331,Z 232.821,A -85,B 0,C 180,E1 -1608.959,E2 -1608.959} C_VEL
LIN {X 0,Y 587.319,Z 232.825,A -85,B 0,C 180,E1 -1611.741,E2 -1611.741} C_VEL
LIN {X 0,Y 587.3,Z 232.826,A -85,B 0,C 180,E1 -1613.814,E2 -1613.814} C_VEL
LIN {X 0,Y 587.289,Z 232.826,A -85,B 0,C 180,E1 -1615.879,E2 -1615.879} C_VEL
LIN {X 0,Y 587.339,Z 232.819,A -85,B 0,C 180,E1 -1617.939,E2 -1617.939} C_VEL
LIN {X 0,Y 587.352,Z 232.817,A -85,B 0,C 180,E1 -1619.996,E2 -1619.996} C_VEL
LIN {X 0,Y 587.345,Z 232.82,A -85,B 0,C 180,E1 -1622.739,E2 -1622.739} C_VEL
LIN {X 0,Y 587.345,Z 232.821,A -85,B 0,C 180,E1 -1625.489,E2 -1625.489} C_VEL
LIN {X 0,Y 587.303,Z 232.823,A -85,B 0,C 180,E1 -1628.252,E2 -1628.252} C_VEL
LIN {X 0,Y 587.372,Z 232.821,A -85,B 0,C 180,E1 -1631.151,E2 -1631.151} C_VEL
LIN {X 0,Y 587.331,Z 232.82,A -85,B 0,C 180,E1 -1634.252,E2 -1634.252} C_VEL
LIN {X 0,Y 587.32,Z 232.822,A -85,B 0,C 180,E1 -1637.402,E2 -1637.402} C_VEL
LIN {X 0,Y 587.277,Z 232.827,A -85,B 0,C 180,E1 -1638.286,E2 -1638.286} C_VEL
LIN {X 0,Y 586.64,Z 232.914,A -85,B 0,C 180,E1 -1638.858,E2 -1638.858} C_VEL
LIN {X 0,Y 583.822,Z 233.264,A -85,B 0,C 180,E1 -1639.787,E2 -1639.787} C_VEL
LIN {X 0,Y 581.412,Z 233.563,A -85,B 0,C 180,E1 -1640.534,E2 -1640.534} C_VEL
LIN {X 0,Y 580.355,Z 233.692,A -85,B 0,C 180,E1 -1641.111,E2 -1641.111} C_VEL
LIN {X 0,Y 580.259,Z 233.701,A -85,B 0,C 180,E1 -1641.306,E2 -1641.306} C_VEL
LIN {X 0,Y 580.245,Z 233.701,A -85,B 0,C 180,E1 -1643.553,E2 -1643.553} C_VEL
LIN {X 0,Y 580.254,Z 233.701,A -85,B 0,C 180,E1 -1645.845,E2 -1645.845} C_VEL
LIN {X 0,Y 580.272,Z 233.702,A -85,B 0,C 180,E1 -1648.18,E2 -1648.18} C_VEL
LIN {X 0,Y 580.245,Z 233.708,A -85,B 0,C 180,E1 -1650.69,E2 -1650.69} C_VEL
LIN {X 0,Y 580.265,Z 233.699,A -85,B 0,C 180,E1 -1653.313,E2 -1653.313} C_VEL
LIN {X 0,Y 580.283,Z 233.698,A -85,B 0,C 180,E1 -1655.763,E2 -1655.763} C_VEL
LIN {X 0,Y 580.246,Z 233.709,A -85,B 0,C 180,E1 -1658.142,E2 -1658.142} C_VEL
LIN {X 0,Y 580.275,Z 233.699,A -85,B 0,C 180,E1 -1660.837,E2 -1660.837} C_VEL
LIN {X 0,Y 580.249,Z 233.704,A -85,B 0,C 180,E1 -1663.652,E2 -1663.652} C_VEL
LIN {X 0,Y 580.232,Z 233.705,A -85,B 0,C 180,E1 -1666.604,E2 -1666.604} C_VEL
LIN {X 0,Y 580.266,Z 233.699,A -85,B 0,C 180,E1 -1669.155,E2 -1669.155} C_VEL
LIN {X 0,Y 580.256,Z 233.71,A -85,B 0,C 180,E1 -1671.92,E2 -1671.92} C_VEL
LIN {X 0,Y 580.251,Z 233.703,A -85,B 0,C 180,E1 -1674.454,E2 -1674.454} C_VEL
LIN {X 0,Y 580.24,Z 233.702,A -85,B 0,C 180,E1 -1676.973,E2 -1676.973} C_VEL
LIN {X 0,Y 580.267,Z 233.703,A -85,B 0,C 180,E1 -1679.424,E2 -1679.424} C_VEL
LIN {X 0,Y 580.259,Z 233.703,A -85,B 0,C 180,E1 -1682.133,E2 -1682.133} C_VEL
LIN {X 0,Y 580.255,Z 233.701,A -85,B 0,C 180,E1 -1684.919,E2 -1684.919} C_VEL
LIN {X 0,Y 580.29,Z 233.7,A -85,B 0,C 180,E1 -1687.198,E2 -1687.198} C_VEL
LIN {X 0,Y 580.255,Z 233.701,A -85,B 0,C 180,E1 -1690.176,E2 -1690.176} C_VEL
LIN {X 0,Y 580.279,Z 233.703,A -85,B 0,C 180,E1 -1693.102,E2 -1693.102} C_VEL
LIN {X 0,Y 580.267,Z 233.701,A -85,B 0,C 180,E1 -1695.982,E2 -1695.982} C_VEL
LIN {X 0,Y 580.279,Z 233.701,A -85,B 0,C 180,E1 -1698.827,E2 -1698.827} C_VEL
LIN {X 0,Y 580.281,Z 233.701,A -85,B 0,C 180,E1 -1701.643,E2 -1701.643} C_VEL
LIN {X 0,Y 580.231,Z 233.706,A -85,B 0,C 180,E1 -1703.742,E2 -1703.742} C_VEL
LIN {X 0,Y 580.21,Z 233.707,A -85,B 0,C 180,E1 -1705.832,E2 -1705.832} C_VEL
LIN {X 0,Y 580.268,Z 233.699,A -85,B 0,C 180,E1 -1707.918,E2 -1707.918} C_VEL
LIN {X 0,Y 580.314,Z 233.699,A -85,B 0,C 180,E1 -1710.694,E2 -1710.694} C_VEL
LIN {X 0,Y 580.237,Z 233.705,A -85,B 0,C 180,E1 -1713.472,E2 -1713.472} C_VEL
LIN {X 0,Y 580.269,Z 233.7,A -85,B 0,C 180,E1 -1715.56,E2 -1715.56} C_VEL
LIN {X 0,Y 580.274,Z 233.699,A -85,B 0,C 180,E1 -1717.656,E2 -1717.656} C_VEL
LIN {X 0,Y 580.253,Z 233.707,A -85,B 0,C 180,E1 -1720.467,E2 -1720.467} C_VEL
LIN {X 0,Y 580.238,Z 233.704,A -85,B 0,C 180,E1 -1723.305,E2 -1723.305} C_VEL
LIN {X 0,Y 580.24,Z 233.706,A -85,B 0,C 180,E1 -1726.175,E2 -1726.175} C_VEL
LIN {X 0,Y 580.267,Z 233.701,A -85,B 0,C 180,E1 -1729.087,E2 -1729.087} C_VEL
LIN {X 0,Y 580.237,Z 233.706,A -85,B 0,C 180,E1 -1732.053,E2 -1732.053} C_VEL
LIN {X 0,Y 580.274,Z 233.702,A -85,B 0,C 180,E1 -1734.737,E2 -1734.737} C_VEL
LIN {X 0,Y 580.23,Z 233.703,A -85,B 0,C 180,E1 -1737.404,E2 -1737.404} C_VEL
LIN {X 0,Y 580.258,Z 233.703,A -85,B 0,C 180,E1 -1739.774,E2 -1739.774} C_VEL
LIN {X 0,Y 580.25,Z 233.711,A -85,B 0,C 180,E1 -1742.203,E2 -1742.203} C_VEL
LIN {X 0,Y 580.245,Z 233.703,A -85,B 0,C 180,E1 -1744.698,E2 -1744.698} C_VEL
LIN {X 0,Y 580.246,Z 233.702,A -85,B 0,C 180,E1 -1747.271,E2 -1747.271} C_VEL
LIN {X 0,Y 580.259,Z 233.705,A -85,B 0,C 180,E1 -1750.277,E2 -1750.277} C_VEL
LIN {X 0,Y 580.236,Z 233.703,A -85,B 0,C 180,E1 -1752.709,E2 -1752.709} C_VEL
LIN {X 0,Y 580.237,Z 233.708,A -85,B 0,C 180,E1 -1755.611,E2 -1755.611} C_VEL
LIN {X 0,Y 580.272,Z 233.701,A -85,B 0,C 180,E1 -1758.239,E2 -1758.239} C_VEL
LIN {X 0,Y 580.238,Z 233.703,A -85,B 0,C 180,E1 -1760.97,E2 -1760.97} C_VEL
LIN {X 0,Y 580.254,Z 233.71,A -85,B 0,C 180,E1 -1763.603,E2 -1763.603} C_VEL
LIN {X 0,Y 580.281,Z 233.699,A -85,B 0,C 180,E1 -1766.15,E2 -1766.15} C_VEL
LIN {X 0,Y 580.241,Z 233.702,A -85,B 0,C 180,E1 -1768.619,E2 -1768.619} C_VEL
LIN {X 0,Y 580.265,Z 233.702,A -85,B 0,C 180,E1 -1771.029,E2 -1771.029} C_VEL
LIN {X 0,Y 580.255,Z 233.706,A -85,B 0,C 180,E1 -1773.671,E2 -1773.671} C_VEL
LIN {X 0,Y 580.266,Z 233.704,A -85,B 0,C 180,E1 -1775.688,E2 -1775.688} C_VEL
LIN {X 0,Y 580.241,Z 233.703,A -85,B 0,C 180,E1 -1777.952,E2 -1777.952} C_VEL
LIN {X 0,Y 580.291,Z 233.701,A -85,B 0,C 180,E1 -1780.919,E2 -1780.919} C_VEL
LIN {X 0,Y 580.249,Z 233.702,A -85,B 0,C 180,E1 -1783.83,E2 -1783.83} C_VEL
LIN {X 0,Y 580.293,Z 233.696,A -85,B 0,C 180,E1 -1785.987,E2 -1785.987} C_VEL
LIN {X 0,Y 580.331,Z 233.697,A -85,B 0,C 180,E1 -1788.832,E2 -1788.832} C_VEL
LIN {X 0,Y 580.277,Z 233.699,A -85,B 0,C 180,E1 -1791.648,E2 -1791.648} C_VEL
LIN {X 0,Y 580.307,Z 233.697,A -85,B 0,C 180,E1 -1794.445,E2 -1794.445} C_VEL
LIN {X 0,Y 580.314,Z 233.697,A -85,B 0,C 180,E1 -1797.228,E2 -1797.228} C_VEL
LIN {X 0,Y 580.323,Z 233.692,A -85,B 0,C 180,E1 -1800.004,E2 -1800.004} C_VEL
LIN {X 0,Y 580.327,Z 233.7,A -85,B 0,C 180,E1 -1802.78,E2 -1802.78} C_VEL
LIN {X 0,Y 580.292,Z 233.696,A -85,B 0,C 180,E1 -1805.564,E2 -1805.564} C_VEL
LIN {X 0,Y 580.252,Z 233.701,A -85,B 0,C 180,E1 -1807.66,E2 -1807.66} C_VEL
LIN {X 0,Y 580.284,Z 233.706,A -85,B 0,C 180,E1 -1810.47,E2 -1810.47} C_VEL
LIN {X 0,Y 580.255,Z 233.7,A -85,B 0,C 180,E1 -1813.308,E2 -1813.308} C_VEL
LIN {X 0,Y 580.278,Z 233.697,A -85,B 0,C 180,E1 -1815.456,E2 -1815.456} C_VEL
LIN {X 0,Y 580.26,Z 233.701,A -85,B 0,C 180,E1 -1817.629,E2 -1817.629} C_VEL
LIN {X 0,Y 580.277,Z 233.701,A -85,B 0,C 180,E1 -1819.826,E2 -1819.826} C_VEL
LIN {X 0,Y 580.262,Z 233.707,A -85,B 0,C 180,E1 -1822.056,E2 -1822.056} C_VEL
LIN {X 0,Y 580.3,Z 233.695,A -85,B 0,C 180,E1 -1825.083,E2 -1825.083} C_VEL
LIN {X 0,Y 580.274,Z 233.706,A -85,B 0,C 180,E1 -1828.19,E2 -1828.19} C_VEL
LIN {X 0,Y 580.27,Z 233.699,A -85,B 0,C 180,E1 -1830.694,E2 -1830.694} C_VEL
LIN {X 0,Y 580.301,Z 233.696,A -85,B 0,C 180,E1 -1833.318,E2 -1833.318} C_VEL
LIN {X 0,Y 580.231,Z 233.711,A -85,B 0,C 180,E1 -1835.756,E2 -1835.756} C_VEL
LIN {X 0,Y 580.283,Z 233.703,A -85,B 0,C 180,E1 -1838.149,E2 -1838.149} C_VEL
LIN {X 0,Y 580.295,Z 233.697,A -85,B 0,C 180,E1 -1840.846,E2 -1840.846} C_VEL
LIN {X 0,Y 580.271,Z 233.708,A -85,B 0,C 180,E1 -1843.661,E2 -1843.661} C_VEL
LIN {X 0,Y 580.253,Z 233.71,A -85,B 0,C 180,E1 -1845.613,E2 -1845.613} C_VEL
LIN {X 0,Y 580.29,Z 233.962,A -85,B 0,C 180,E1 -1846.345,E2 -1846.345} C_VEL
LIN {X 0,Y 580.509,Z 236.946,A -85,B 0,C 180,E1 -1848.253,E2 -1848.253} C_VEL
LIN {X 0,Y 580.505,Z 241.596,A -85,B 0,C 180,E1 -1850.984,E2 -1850.984} C_VEL
LIN {X 0,Y 580.447,Z 246.374,A -85,B 0,C 180,E1 -1853.61,E2 -1853.61} C_VEL
LIN {X 0,Y 580.373,Z 251.306,A -85,B 0,C 180,E1 -1856.15,E2 -1856.15} C_VEL
LIN {X 0,Y 580.317,Z 256.354,A -85,B 0,C 180,E1 -1858.618,E2 -1858.618} C_VEL
LIN {X 0,Y 580.245,Z 261.47,A -85,B 0,C 180,E1 -1861.022,E2 -1861.022} C_VEL
LIN {X 0,Y 580.242,Z 267.475,A -85,B 0,C 180,E1 -1863.678,E2 -1863.678} C_VEL
LIN {X 0,Y 580.171,Z 273.903,A -85,B 0,C 180,E1 -1866.438,E2 -1866.438} C_VEL
LIN {X 0,Y 580.176,Z 279.721,A -85,B 0,C 180,E1 -1868.869,E2 -1868.869} C_VEL
LIN {X 0,Y 580.142,Z 286.478,A -85,B 0,C 180,E1 -1871.641,E2 -1871.641} C_VEL
LIN {X 0,Y 580.111,Z 293.664,A -85,B 0,C 180,E1 -1874.543,E2 -1874.543} C_VEL
LIN {X 0,Y 580.08,Z 299.054,A -85,B 0,C 180,E1 -1876.692,E2 -1876.692} C_VEL
LIN {X 0,Y 580.078,Z 301.524,A -85,B 0,C 180,E1 -1877.671,E2 -1877.671} C_VEL
LIN {X 0,Y 580.777,Z 307.543,A -85,B 0,C 180,E1 -1877.796,E2 -1877.796} C_VEL
LIN {X 0,Y 580.712,Z 319.812,A -85,B 0,C 180,E1 -1878.127,E2 -1878.127} C_VEL
LIN {X 0,Y 580.574,Z 331.705,A -85,B 0,C 180,E1 -1878.578,E2 -1878.578} C_VEL
LIN {X 0,Y 580.502,Z 342.189,A -85,B 0,C 180,E1 -1879.096,E2 -1879.096} C_VEL
LIN {X 0,Y 580.439,Z 353.487,A -85,B 0,C 180,E1 -1879.801,E2 -1879.801} C_VEL
LIN {X 0,Y 580.352,Z 363.638,A -85,B 0,C 180,E1 -1880.591,E2 -1880.591} C_VEL
LIN {X 0,Y 580.27,Z 372.757,A -85,B 0,C 180,E1 -1881.468,E2 -1881.468} C_VEL
LIN {X 0,Y 580.221,Z 380.304,A -85,B 0,C 180,E1 -1882.343,E2 -1882.343} C_VEL
LIN {X 0,Y 580.134,Z 387.85,A -85,B 0,C 180,E1 -1883.41,E2 -1883.41} C_VEL
LIN {X 0,Y 580.138,Z 393.683,A -85,B 0,C 180,E1 -1884.439,E2 -1884.439} C_VEL
LIN {X 0,Y 580.108,Z 398.38,A -85,B 0,C 180,E1 -1885.484,E2 -1885.484} C_VEL
LIN {X 0,Y 580.123,Z 401.967,A -85,B 0,C 180,E1 -1886.527,E2 -1886.527} C_VEL
LIN {X 0,Y 580.043,Z 403.79,A -85,B 0,C 180,E1 -1887.222,E2 -1887.222} C_VEL
LIN {X 0,Y 580.047,Z 406.19,A -85,B 0,C 180,E1 -1888.611,E2 -1888.611} C_VEL
LIN {X 0,Y 580.04,Z 406.782,A -85,B 0,C 180,E1 -1889.306,E2 -1889.306} C_VEL
LIN {X 0,Y 580.04,Z 406.782,A -85,B 0,C 180,E1 -1890.694,E2 -1890.694} C_VEL
LIN {X 0,Y 580.047,Z 406.19,A -85,B 0,C 180,E1 -1891.389,E2 -1891.389} C_VEL
LIN {X 0,Y 580.043,Z 403.79,A -85,B 0,C 180,E1 -1892.778,E2 -1892.778} C_VEL
LIN {X 0,Y 580.11,Z 400.876,A -85,B 0,C 180,E1 -1893.82,E2 -1893.82} C_VEL
LIN {X 0,Y 580.053,Z 396.925,A -85,B 0,C 180,E1 -1894.865,E2 -1894.865} C_VEL
LIN {X 0,Y 580.162,Z 391.83,A -85,B 0,C 180,E1 -1895.91,E2 -1895.91} C_VEL
LIN {X 0,Y 580.159,Z 385.446,A -85,B 0,C 180,E1 -1896.958,E2 -1896.958} C_VEL
LIN {X 0,Y 580.243,Z 377.493,A -85,B 0,C 180,E1 -1898.007,E2 -1898.007} C_VEL
LIN {X 0,Y 580.305,Z 369.353,A -85,B 0,C 180,E1 -1898.883,E2 -1898.883} C_VEL
LIN {X 0,Y 580.357,Z 359.349,A -85,B 0,C 180,E1 -1899.761,E2 -1899.761} C_VEL
LIN {X 0,Y 580.446,Z 349.527,A -85,B 0,C 180,E1 -1900.464,E2 -1900.464} C_VEL
LIN {X 0,Y 580.525,Z 338.93,A -85,B 0,C 180,E1 -1901.08,E2 -1901.08} C_VEL
LIN {X 0,Y 580.631,Z 326.162,A -85,B 0,C 180,E1 -1901.653,E2 -1901.653} C_VEL
LIN {X 0,Y 580.771,Z 313.828,A -85,B 0,C 180,E1 -1902.049,E2 -1902.049} C_VEL
LIN {X 0,Y 580.695,Z 305.285,A -85,B 0,C 180,E1 -1902.25,E2 -1902.25} C_VEL
LIN {X 0,Y 580.078,Z 301.524,A -85,B 0,C 180,E1 -1902.329,E2 -1902.329} C_VEL
LIN {X 0,Y 580.122,Z 295.461,A -85,B 0,C 180,E1 -1904.738,E2 -1904.738} C_VEL
LIN {X 0,Y 580.145,Z 288.275,A -85,B 0,C 180,E1 -1907.629,E2 -1907.629} C_VEL
LIN {X 0,Y 580.157,Z 282.885,A -85,B 0,C 180,E1 -1909.827,E2 -1909.827} C_VEL
LIN {X 0,Y 580.194,Z 277.496,A -85,B 0,C 180,E1 -1912.055,E2 -1912.055} C_VEL
LIN {X 0,Y 580.191,Z 270.341,A -85,B 0,C 180,E1 -1915.084,E2 -1915.084} C_VEL
LIN {X 0,Y 580.24,Z 263.998,A -85,B 0,C 180,E1 -1917.846,E2 -1917.846} C_VEL
LIN {X 0,Y 580.3,Z 257.804,A -85,B 0,C 180,E1 -1920.695,E2 -1920.695} C_VEL
LIN {X 0,Y 580.381,Z 252.34,A -85,B 0,C 180,E1 -1923.326,E2 -1923.326} C_VEL
LIN {X 0,Y 580.428,Z 247.533,A -85,B 0,C 180,E1 -1925.779,E2 -1925.779} C_VEL
LIN {X 0,Y 580.463,Z 243.153,A -85,B 0,C 180,E1 -1928.132,E2 -1928.132} C_VEL
LIN {X 0,Y 580.497,Z 239.365,A -85,B 0,C 180,E1 -1930.292,E2 -1930.292} C_VEL
LIN {X 0,Y 580.479,Z 235.445,A -85,B 0,C 180,E1 -1932.687,E2 -1932.687} C_VEL
LIN {X 0,Y 580.29,Z 233.954,A -85,B 0,C 180,E1 -1933.655,E2 -1933.655} C_VEL
LIN {X 0,Y 580.258,Z 233.704,A -85,B 0,C 180,E1 -1935.609,E2 -1935.609} C_VEL
LIN {X 0,Y 580.273,Z 233.703,A -85,B 0,C 180,E1 -1938.668,E2 -1938.668} C_VEL
LIN {X 0,Y 580.266,Z 233.7,A -85,B 0,C 180,E1 -1940.962,E2 -1940.962} C_VEL
LIN {X 0,Y 580.245,Z 233.705,A -85,B 0,C 180,E1 -1943.592,E2 -1943.592} C_VEL
LIN {X 0,Y 580.309,Z 233.703,A -85,B 0,C 180,E1 -1946.142,E2 -1946.142} C_VEL
LIN {X 0,Y 580.266,Z 233.7,A -85,B 0,C 180,E1 -1948.611,E2 -1948.611} C_VEL
LIN {X 0,Y 580.283,Z 233.697,A -85,B 0,C 180,E1 -1951.021,E2 -1951.021} C_VEL
LIN {X 0,Y 580.26,Z 233.705,A -85,B 0,C 180,E1 -1954.147,E2 -1954.147} C_VEL
LIN {X 0,Y 580.268,Z 233.7,A -85,B 0,C 180,E1 -1956.439,E2 -1956.439} C_VEL
LIN {X 0,Y 580.264,Z 233.704,A -85,B 0,C 180,E1 -1959.434,E2 -1959.434} C_VEL
LIN {X 0,Y 580.248,Z 233.71,A -85,B 0,C 180,E1 -1961.641,E2 -1961.641} C_VEL
LIN {X 0,Y 580.253,Z 233.707,A -85,B 0,C 180,E1 -1963.822,E2 -1963.822} C_VEL
LIN {X 0,Y 580.315,Z 233.697,A -85,B 0,C 180,E1 -1965.98,E2 -1965.98} C_VEL
LIN {X 0,Y 580.299,Z 233.696,A -85,B 0,C 180,E1 -1968.823,E2 -1968.823} C_VEL
LIN {X 0,Y 580.291,Z 233.702,A -85,B 0,C 180,E1 -1971.64,E2 -1971.64} C_VEL
LIN {X 0,Y 580.261,Z 233.704,A -85,B 0,C 180,E1 -1973.738,E2 -1973.738} C_VEL
LIN {X 0,Y 580.246,Z 233.704,A -85,B 0,C 180,E1 -1975.829,E2 -1975.829} C_VEL
LIN {X 0,Y 580.312,Z 233.695,A -85,B 0,C 180,E1 -1977.914,E2 -1977.914} C_VEL
LIN {X 0,Y 580.323,Z 233.692,A -85,B 0,C 180,E1 -1979.996,E2 -1979.996} C_VEL
LIN {X 0,Y 580.314,Z 233.697,A -85,B 0,C 180,E1 -1982.772,E2 -1982.772} C_VEL
LIN {X 0,Y 580.307,Z 233.697,A -85,B 0,C 180,E1 -1985.555,E2 -1985.555} C_VEL
LIN {X 0,Y 580.277,Z 233.699,A -85,B 0,C 180,E1 -1988.352,E2 -1988.352} C_VEL
LIN {X 0,Y 580.319,Z 233.698,A -85,B 0,C 180,E1 -1991.206,E2 -1991.206} C_VEL
LIN {X 0,Y 580.284,Z 233.699,A -85,B 0,C 180,E1 -1994.331,E2 -1994.331} C_VEL
LIN {X 0,Y 580.286,Z 233.705,A -85,B 0,C 180,E1 -1996.909,E2 -1996.909} C_VEL
LIN {X 0,Y 580.277,Z 233.698,A -85,B 0,C 180,E1 -1999.818,E2 -1999.818} C_VEL
LIN {X 0,Y 580.259,Z 233.701,A -85,B 0,C 180,E1 -2001.306,E2 -2001.306} C_VEL
LIN {X 0,Y 579.557,Z 233.789,A -85,B 0,C 180,E1 -2001.885,E2 -2001.885} C_VEL
LIN {X 0,Y 576.677,Z 234.153,A -85,B 0,C 180,E1 -2002.825,E2 -2002.825} C_VEL
LIN {X 0,Y 574.281,Z 234.448,A -85,B 0,C 180,E1 -2003.581,E2 -2003.581} C_VEL
LIN {X 0,Y 573.281,Z 234.572,A -85,B 0,C 180,E1 -2004.165,E2 -2004.165} C_VEL
LIN {X 0,Y 573.214,Z 234.583,A -85,B 0,C 180,E1 -2004.363,E2 -2004.363} C_VEL
LIN {X 0,Y 573.216,Z 234.581,A -85,B 0,C 180,E1 -2006.971,E2 -2006.971} C_VEL
LIN {X 0,Y 573.212,Z 234.578,A -85,B 0,C 180,E1 -2009.484,E2 -2009.484} C_VEL
LIN {X 0,Y 573.218,Z 234.583,A -85,B 0,C 180,E1 -2012.64,E2 -2012.64} C_VEL
LIN {X 0,Y 573.226,Z 234.576,A -85,B 0,C 180,E1 -2015.179,E2 -2015.179} C_VEL
LIN {X 0,Y 573.194,Z 234.583,A -85,B 0,C 180,E1 -2017.803,E2 -2017.803} C_VEL
LIN {X 0,Y 573.221,Z 234.582,A -85,B 0,C 180,E1 -2020.524,E2 -2020.524} C_VEL
LIN {X 0,Y 573.208,Z 234.578,A -85,B 0,C 180,E1 -2023.353,E2 -2023.353} C_VEL
LIN {X 0,Y 573.2,Z 234.585,A -85,B 0,C 180,E1 -2026.326,E2 -2026.326} C_VEL
LIN {X 0,Y 573.206,Z 234.581,A -85,B 0,C 180,E1 -2028.542,E2 -2028.542} C_VEL
LIN {X 0,Y 573.199,Z 234.58,A -85,B 0,C 180,E1 -2031.296,E2 -2031.296} C_VEL
LIN {X 0,Y 573.207,Z 234.586,A -85,B 0,C 180,E1 -2034.007,E2 -2034.007} C_VEL
LIN {X 0,Y 573.224,Z 234.577,A -85,B 0,C 180,E1 -2036.516,E2 -2036.516} C_VEL
LIN {X 0,Y 573.197,Z 234.581,A -85,B 0,C 180,E1 -2039.109,E2 -2039.109} C_VEL
LIN {X 0,Y 573.213,Z 234.583,A -85,B 0,C 180,E1 -2041.435,E2 -2041.435} C_VEL
LIN {X 0,Y 573.23,Z 234.583,A -85,B 0,C 180,E1 -2043.809,E2 -2043.809} C_VEL
LIN {X 0,Y 573.243,Z 234.574,A -85,B 0,C 180,E1 -2046.835,E2 -2046.835} C_VEL
LIN {X 0,Y 573.205,Z 234.582,A -85,B 0,C 180,E1 -2049.922,E2 -2049.922} C_VEL
LIN {X 0,Y 573.241,Z 234.578,A -85,B 0,C 180,E1 -2052.971,E2 -2052.971} C_VEL
LIN {X 0,Y 573.214,Z 234.581,A -85,B 0,C 180,E1 -2055.806,E2 -2055.806} C_VEL
LIN {X 0,Y 573.212,Z 234.58,A -85,B 0,C 180,E1 -2058.733,E2 -2058.733} C_VEL
LIN {X 0,Y 573.255,Z 234.578,A -85,B 0,C 180,E1 -2061.54,E2 -2061.54} C_VEL
LIN {X 0,Y 573.194,Z 234.583,A -85,B 0,C 180,E1 -2063.665,E2 -2063.665} C_VEL
LIN {X 0,Y 573.169,Z 234.585,A -85,B 0,C 180,E1 -2065.781,E2 -2065.781} C_VEL
LIN {X 0,Y 573.239,Z 234.575,A -85,B 0,C 180,E1 -2067.892,E2 -2067.892} C_VEL
LIN {X 0,Y 573.282,Z 234.575,A -85,B 0,C 180,E1 -2070.702,E2 -2070.702} C_VEL
LIN {X 0,Y 573.188,Z 234.583,A -85,B 0,C 180,E1 -2073.515,E2 -2073.515} C_VEL
LIN {X 0,Y 573.236,Z 234.576,A -85,B 0,C 180,E1 -2075.629,E2 -2075.629} C_VEL
LIN {X 0,Y 573.226,Z 234.577,A -85,B 0,C 180,E1 -2077.751,E2 -2077.751} C_VEL
LIN {X 0,Y 573.222,Z 234.585,A -85,B 0,C 180,E1 -2080.597,E2 -2080.597} C_VEL
LIN {X 0,Y 573.192,Z 234.581,A -85,B 0,C 180,E1 -2083.471,E2 -2083.471} C_VEL
LIN {X 0,Y 573.212,Z 234.585,A -85,B 0,C 180,E1 -2086.379,E2 -2086.379} C_VEL
LIN {X 0,Y 573.209,Z 234.578,A -85,B 0,C 180,E1 -2089.332,E2 -2089.332} C_VEL
LIN {X 0,Y 573.21,Z 234.586,A -85,B 0,C 180,E1 -2092.338,E2 -2092.338} C_VEL
LIN {X 0,Y 573.219,Z 234.579,A -85,B 0,C 180,E1 -2094.885,E2 -2094.885} C_VEL
LIN {X 0,Y 573.228,Z 234.578,A -85,B 0,C 180,E1 -2097.767,E2 -2097.767} C_VEL
LIN {X 0,Y 573.214,Z 234.586,A -85,B 0,C 180,E1 -2100.177,E2 -2100.177} C_VEL
LIN {X 0,Y 573.203,Z 234.582,A -85,B 0,C 180,E1 -2102.647,E2 -2102.647} C_VEL
LIN {X 0,Y 573.212,Z 234.578,A -85,B 0,C 180,E1 -2105.187,E2 -2105.187} C_VEL
LIN {X 0,Y 573.195,Z 234.585,A -85,B 0,C 180,E1 -2107.81,E2 -2107.81} C_VEL
LIN {X 0,Y 573.213,Z 234.58,A -85,B 0,C 180,E1 -2110.532,E2 -2110.532} C_VEL
LIN {X 0,Y 573.194,Z 234.582,A -85,B 0,C 180,E1 -2113.362,E2 -2113.362} C_VEL
LIN {X 0,Y 573.213,Z 234.58,A -85,B 0,C 180,E1 -2116.333,E2 -2116.333} C_VEL
LIN {X 0,Y 573.212,Z 234.578,A -85,B 0,C 180,E1 -2118.55,E2 -2118.55} C_VEL
LIN {X 0,Y 573.201,Z 234.582,A -85,B 0,C 180,E1 -2121.303,E2 -2121.303} C_VEL
LIN {X 0,Y 573.221,Z 234.581,A -85,B 0,C 180,E1 -2124.015,E2 -2124.015} C_VEL
LIN {X 0,Y 573.244,Z 234.574,A -85,B 0,C 180,E1 -2126.523,E2 -2126.523} C_VEL
LIN {X 0,Y 573.191,Z 234.584,A -85,B 0,C 180,E1 -2129.122,E2 -2129.122} C_VEL
LIN {X 0,Y 573.232,Z 234.578,A -85,B 0,C 180,E1 -2131.972,E2 -2131.972} C_VEL
LIN {X 0,Y 573.217,Z 234.577,A -85,B 0,C 180,E1 -2134.594,E2 -2134.594} C_VEL
LIN {X 0,Y 573.206,Z 234.583,A -85,B 0,C 180,E1 -2137.667,E2 -2137.667} C_VEL
LIN {X 0,Y 573.227,Z 234.577,A -85,B 0,C 180,E1 -2139.928,E2 -2139.928} C_VEL
LIN {X 0,Y 573.233,Z 234.582,A -85,B 0,C 180,E1 -2142.995,E2 -2142.995} C_VEL
LIN {X 0,Y 573.241,Z 234.575,A -85,B 0,C 180,E1 -2145.811,E2 -2145.811} C_VEL
LIN {X 0,Y 573.268,Z 234.576,A -85,B 0,C 180,E1 -2148.736,E2 -2148.736} C_VEL
LIN {X 0,Y 573.224,Z 234.578,A -85,B 0,C 180,E1 -2151.544,E2 -2151.544} C_VEL
LIN {X 0,Y 573.194,Z 234.58,A -85,B 0,C 180,E1 -2153.669,E2 -2153.669} C_VEL
LIN {X 0,Y 573.189,Z 234.58,A -85,B 0,C 180,E1 -2155.785,E2 -2155.785} C_VEL
LIN {X 0,Y 573.277,Z 234.57,A -85,B 0,C 180,E1 -2157.897,E2 -2157.897} C_VEL
LIN {X 0,Y 573.329,Z 234.572,A -85,B 0,C 180,E1 -2160.706,E2 -2160.706} C_VEL
LIN {X 0,Y 573.291,Z 234.576,A -85,B 0,C 180,E1 -2162.815,E2 -2162.815} C_VEL
LIN {X 0,Y 573.261,Z 234.572,A -85,B 0,C 180,E1 -2165.632,E2 -2165.632} C_VEL
LIN {X 0,Y 573.208,Z 234.578,A -85,B 0,C 180,E1 -2167.755,E2 -2167.755} C_VEL
LIN {X 0,Y 573.253,Z 234.581,A -85,B 0,C 180,E1 -2170.6,E2 -2170.6} C_VEL
LIN {X 0,Y 573.216,Z 234.577,A -85,B 0,C 180,E1 -2173.474,E2 -2173.474} C_VEL
LIN {X 0,Y 573.217,Z 234.578,A -85,B 0,C 180,E1 -2175.652,E2 -2175.652} C_VEL
LIN {X 0,Y 573.219,Z 234.58,A -85,B 0,C 180,E1 -2177.852,E2 -2177.852} C_VEL
LIN {X 0,Y 573.233,Z 234.582,A -85,B 0,C 180,E1 -2180.08,E2 -2180.08} C_VEL
LIN {X 0,Y 573.227,Z 234.583,A -85,B 0,C 180,E1 -2182.341,E2 -2182.341} C_VEL
LIN {X 0,Y 573.238,Z 234.575,A -85,B 0,C 180,E1 -2185.414,E2 -2185.414} C_VEL
LIN {X 0,Y 573.22,Z 234.579,A -85,B 0,C 180,E1 -2188.568,E2 -2188.568} C_VEL
LIN {X 0,Y 573.218,Z 234.577,A -85,B 0,C 180,E1 -2190.996,E2 -2190.996} C_VEL
LIN {X 0,Y 573.265,Z 234.575,A -85,B 0,C 180,E1 -2193.526,E2 -2193.526} C_VEL
LIN {X 0,Y 573.19,Z 234.588,A -85,B 0,C 180,E1 -2196.056,E2 -2196.056} C_VEL
LIN {X 0,Y 573.235,Z 234.576,A -85,B 0,C 180,E1 -2198.705,E2 -2198.705} C_VEL
LIN {X 0,Y 573.222,Z 234.586,A -85,B 0,C 180,E1 -2201.594,E2 -2201.594} C_VEL
LIN {X 0,Y 573.225,Z 234.581,A -85,B 0,C 180,E1 -2204.337,E2 -2204.337} C_VEL
LIN {X 0,Y 573.221,Z 234.586,A -85,B 0,C 180,E1 -2205.667,E2 -2205.667} C_VEL
LIN {X 0,Y 573.384,Z 235.689,A -85,B 0,C 180,E1 -2206.656,E2 -2206.656} C_VEL
LIN {X 0,Y 573.525,Z 238.687,A -85,B 0,C 180,E1 -2208.57,E2 -2208.57} C_VEL
LIN {X 0,Y 573.476,Z 243.355,A -85,B 0,C 180,E1 -2211.318,E2 -2211.318} C_VEL
LIN {X 0,Y 573.414,Z 248.202,A -85,B 0,C 180,E1 -2213.993,E2 -2213.993} C_VEL
LIN {X 0,Y 573.366,Z 253.109,A -85,B 0,C 180,E1 -2216.525,E2 -2216.525} C_VEL
LIN {X 0,Y 573.261,Z 258.37,A -85,B 0,C 180,E1 -2219.115,E2 -2219.115} C_VEL
LIN {X 0,Y 573.195,Z 264.488,A -85,B 0,C 180,E1 -2221.984,E2 -2221.984} C_VEL
LIN {X 0,Y 573.133,Z 270.344,A -85,B 0,C 180,E1 -2224.585,E2 -2224.585} C_VEL
LIN {X 0,Y 573.115,Z 275.644,A -85,B 0,C 180,E1 -2226.896,E2 -2226.896} C_VEL
LIN {X 0,Y 573.106,Z 281.089,A -85,B 0,C 180,E1 -2229.169,E2 -2229.169} C_VEL
LIN {X 0,Y 573.071,Z 286.478,A -85,B 0,C 180,E1 -2231.407,E2 -2231.407} C_VEL
LIN {X 0,Y 573.051,Z 291.868,A -85,B 0,C 180,E1 -2233.616,E2 -2233.616} C_VEL
LIN {X 0,Y 573.015,Z 299.054,A -85,B 0,C 180,E1 -2236.525,E2 -2236.525} C_VEL
LIN {X 0,Y 572.992,Z 301.524,A -85,B 0,C 180,E1 -2237.516,E2 -2237.516} C_VEL
LIN {X 0,Y 573.846,Z 307.542,A -85,B 0,C 180,E1 -2237.647,E2 -2237.647} C_VEL
LIN {X 0,Y 573.765,Z 319.796,A -85,B 0,C 180,E1 -2237.982,E2 -2237.982} C_VEL
LIN {X 0,Y 573.644,Z 330.433,A -85,B 0,C 180,E1 -2238.383,E2 -2238.383} C_VEL
LIN {X 0,Y 573.524,Z 340.925,A -85,B 0,C 180,E1 -2238.893,E2 -2238.893} C_VEL
LIN {X 0,Y 573.436,Z 350.861,A -85,B 0,C 180,E1 -2239.496,E2 -2239.496} C_VEL
LIN {X 0,Y 573.341,Z 361.555,A -85,B 0,C 180,E1 -2240.297,E2 -2240.297} C_VEL
LIN {X 0,Y 573.239,Z 371.119,A -85,B 0,C 180,E1 -2241.185,E2 -2241.185} C_VEL
LIN {X 0,Y 573.162,Z 378.926,A -85,B 0,C 180,E1 -2242.071,E2 -2242.071} C_VEL
LIN {X 0,Y 573.084,Z 385.437,A -85,B 0,C 180,E1 -2242.956,E2 -2242.956} C_VEL
LIN {X 0,Y 573.074,Z 391.821,A -85,B 0,C 180,E1 -2244.017,E2 -2244.017} C_VEL
LIN {X 0,Y 572.962,Z 396.917,A -85,B 0,C 180,E1 -2245.074,E2 -2245.074} C_VEL
LIN {X 0,Y 573.015,Z 400.869,A -85,B 0,C 180,E1 -2246.132,E2 -2246.132} C_VEL
LIN {X 0,Y 572.959,Z 403.785,A -85,B 0,C 180,E1 -2247.188,E2 -2247.188} C_VEL
LIN {X 0,Y 572.946,Z 406.192,A -85,B 0,C 180,E1 -2248.594,E2 -2248.594} C_VEL
LIN {X 0,Y 572.941,Z 406.781,A -85,B 0,C 180,E1 -2249.297,E2 -2249.297} C_VEL
LIN {X 0,Y 572.941,Z 406.781,A -85,B 0,C 180,E1 -2250.703,E2 -2250.703} C_VEL
LIN {X 0,Y 572.946,Z 406.192,A -85,B 0,C 180,E1 -2251.406,E2 -2251.406} C_VEL
LIN {X 0,Y 572.959,Z 403.785,A -85,B 0,C 180,E1 -2252.812,E2 -2252.812} C_VEL
LIN {X 0,Y 573.015,Z 400.869,A -85,B 0,C 180,E1 -2253.868,E2 -2253.868} C_VEL
LIN {X 0,Y 572.962,Z 396.917,A -85,B 0,C 180,E1 -2254.926,E2 -2254.926} C_VEL
LIN {X 0,Y 573.075,Z 391.821,A -85,B 0,C 180,E1 -2255.983,E2 -2255.983} C_VEL
LIN {X 0,Y 573.084,Z 385.437,A -85,B 0,C 180,E1 -2257.044,E2 -2257.044} C_VEL
LIN {X 0,Y 573.179,Z 377.497,A -85,B 0,C 180,E1 -2258.106,E2 -2258.106} C_VEL
LIN {X 0,Y 573.28,Z 369.356,A -85,B 0,C 180,E1 -2258.992,E2 -2258.992} C_VEL
LIN {X 0,Y 573.336,Z 359.336,A -85,B 0,C 180,E1 -2259.881,E2 -2259.881} C_VEL
LIN {X 0,Y 573.458,Z 349.512,A -85,B 0,C 180,E1 -2260.593,E2 -2260.593} C_VEL
LIN {X 0,Y 573.558,Z 338.75,A -85,B 0,C 180,E1 -2261.225,E2 -2261.225} C_VEL
LIN {X 0,Y 573.674,Z 326.169,A -85,B 0,C 180,E1 -2261.796,E2 -2261.796} C_VEL
LIN {X 0,Y 573.824,Z 313.796,A -85,B 0,C 180,E1 -2262.197,E2 -2262.197} C_VEL
LIN {X 0,Y 573.658,Z 305.714,A -85,B 0,C 180,E1 -2262.394,E2 -2262.394} C_VEL
LIN {X 0,Y 572.992,Z 301.524,A -85,B 0,C 180,E1 -2262.484,E2 -2262.484} C_VEL
LIN {X 0,Y 573.047,Z 295.461,A -85,B 0,C 180,E1 -2264.924,E2 -2264.924} C_VEL
LIN {X 0,Y 573.083,Z 288.275,A -85,B 0,C 180,E1 -2267.853,E2 -2267.853} C_VEL
LIN {X 0,Y 573.074,Z 282.885,A -85,B 0,C 180,E1 -2270.083,E2 -2270.083} C_VEL
LIN {X 0,Y 573.109,Z 277.476,A -85,B 0,C 180,E1 -2272.342,E2 -2272.342} C_VEL
LIN {X 0,Y 573.151,Z 271.618,A -85,B 0,C 180,E1 -2274.851,E2 -2274.851} C_VEL
LIN {X 0,Y 573.2,Z 265.041,A -85,B 0,C 180,E1 -2277.769,E2 -2277.769} C_VEL
LIN {X 0,Y 573.246,Z 259.847,A -85,B 0,C 180,E1 -2280.175,E2 -2280.175} C_VEL
LIN {X 0,Y 573.315,Z 254.742,A -85,B 0,C 180,E1 -2282.64,E2 -2282.64} C_VEL
LIN {X 0,Y 573.399,Z 249.771,A -85,B 0,C 180,E1 -2285.173,E2 -2285.173} C_VEL
LIN {X 0,Y 573.452,Z 244.91,A -85,B 0,C 180,E1 -2287.79,E2 -2287.79} C_VEL
LIN {X 0,Y 573.506,Z 240.129,A -85,B 0,C 180,E1 -2290.553,E2 -2290.553} C_VEL
LIN {X 0,Y 573.51,Z 236.718,A -85,B 0,C 180,E1 -2292.668,E2 -2292.668} C_VEL
LIN {X 0,Y 573.312,Z 235.197,A -85,B 0,C 180,E1 -2293.674,E2 -2293.674} C_VEL
LIN {X 0,Y 573.221,Z 234.585,A -85,B 0,C 180,E1 -2294.333,E2 -2294.333} C_VEL
LIN {X 0,Y 573.23,Z 234.583,A -85,B 0,C 180,E1 -2296.638,E2 -2296.638} C_VEL
LIN {X 0,Y 573.249,Z 234.575,A -85,B 0,C 180,E1 -2299.473,E2 -2299.473} C_VEL
LIN {X 0,Y 573.229,Z 234.586,A -85,B 0,C 180,E1 -2302.19,E2 -2302.19} C_VEL
LIN {X 0,Y 573.224,Z 234.577,A -85,B 0,C 180,E1 -2305.228,E2 -2305.228} C_VEL
LIN {X 0,Y 573.247,Z 234.579,A -85,B 0,C 180,E1 -2307.77,E2 -2307.77} C_VEL
LIN {X 0,Y 573.241,Z 234.575,A -85,B 0,C 180,E1 -2310.63,E2 -2310.63} C_VEL
LIN {X 0,Y 573.203,Z 234.583,A -85,B 0,C 180,E1 -2313.512,E2 -2313.512} C_VEL
LIN {X 0,Y 573.224,Z 234.581,A -85,B 0,C 180,E1 -2316.131,E2 -2316.131} C_VEL
LIN {X 0,Y 573.245,Z 234.575,A -85,B 0,C 180,E1 -2319.17,E2 -2319.17} C_VEL
LIN {X 0,Y 573.204,Z 234.584,A -85,B 0,C 180,E1 -2321.407,E2 -2321.407} C_VEL
LIN {X 0,Y 573.231,Z 234.585,A -85,B 0,C 180,E1 -2323.618,E2 -2323.618} C_VEL
LIN {X 0,Y 573.265,Z 234.577,A -85,B 0,C 180,E1 -2325.803,E2 -2325.803} C_VEL
LIN {X 0,Y 573.257,Z 234.572,A -85,B 0,C 180,E1 -2328.742,E2 -2328.742} C_VEL
LIN {X 0,Y 573.237,Z 234.583,A -85,B 0,C 180,E1 -2331.536,E2 -2331.536} C_VEL
LIN {X 0,Y 573.224,Z 234.582,A -85,B 0,C 180,E1 -2333.661,E2 -2333.661} C_VEL
LIN {X 0,Y 573.204,Z 234.582,A -85,B 0,C 180,E1 -2335.777,E2 -2335.777} C_VEL
LIN {X 0,Y 573.284,Z 234.57,A -85,B 0,C 180,E1 -2337.888,E2 -2337.888} C_VEL
LIN {X 0,Y 573.294,Z 234.568,A -85,B 0,C 180,E1 -2339.996,E2 -2339.996} C_VEL
LIN {X 0,Y 573.282,Z 234.573,A -85,B 0,C 180,E1 -2342.806,E2 -2342.806} C_VEL
LIN {X 0,Y 573.27,Z 234.573,A -85,B 0,C 180,E1 -2345.624,E2 -2345.624} C_VEL
LIN {X 0,Y 573.25,Z 234.574,A -85,B 0,C 180,E1 -2347.746,E2 -2347.746} C_VEL
LIN {X 0,Y 573.244,Z 234.577,A -85,B 0,C 180,E1 -2350.592,E2 -2350.592} C_VEL
LIN {X 0,Y 573.238,Z 234.581,A -85,B 0,C 180,E1 -2352.744,E2 -2352.744} C_VEL
LIN {X 0,Y 573.211,Z 234.587,A -85,B 0,C 180,E1 -2354.915,E2 -2354.915} C_VEL
LIN {X 0,Y 573.214,Z 234.577,A -85,B 0,C 180,E1 -2357.844,E2 -2357.844} C_VEL
LIN {X 0,Y 573.227,Z 234.577,A -85,B 0,C 180,E1 -2360.072,E2 -2360.072} C_VEL
LIN {X 0,Y 573.206,Z 234.583,A -85,B 0,C 180,E1 -2362.333,E2 -2362.333} C_VEL
LIN {X 0,Y 573.214,Z 234.583,A -85,B 0,C 180,E1 -2364.363,E2 -2364.363} C_VEL
LIN {X 0,Y 572.586,Z 234.667,A -85,B 0,C 180,E1 -2364.949,E2 -2364.949} C_VEL
LIN {X 0,Y 569.747,Z 235.019,A -85,B 0,C 180,E1 -2365.901,E2 -2365.901} C_VEL
LIN {X 0,Y 567.319,Z 235.32,A -85,B 0,C 180,E1 -2366.666,E2 -2366.666} C_VEL
LIN {X 0,Y 566.267,Z 235.444,A -85,B 0,C 180,E1 -2367.257,E2 -2367.257} C_VEL
LIN {X 0,Y 566.178,Z 235.454,A -85,B 0,C 180,E1 -2367.457,E2 -2367.457} C_VEL
LIN {X 0,Y 566.164,Z 235.456,A -85,B 0,C 180,E1 -2369.764,E2 -2369.764} C_VEL
LIN {X 0,Y 566.17,Z 235.465,A -85,B 0,C 180,E1 -2372.427,E2 -2372.427} C_VEL
LIN {X 0,Y 566.172,Z 235.456,A -85,B 0,C 180,E1 -2374.99,E2 -2374.99} C_VEL
LIN {X 0,Y 566.153,Z 235.457,A -85,B 0,C 180,E1 -2377.456,E2 -2377.456} C_VEL
LIN {X 0,Y 566.18,Z 235.463,A -85,B 0,C 180,E1 -2380.193,E2 -2380.193} C_VEL
LIN {X 0,Y 566.165,Z 235.456,A -85,B 0,C 180,E1 -2383.049,E2 -2383.049} C_VEL
LIN {X 0,Y 566.15,Z 235.467,A -85,B 0,C 180,E1 -2386.044,E2 -2386.044} C_VEL
LIN {X 0,Y 566.166,Z 235.456,A -85,B 0,C 180,E1 -2388.861,E2 -2388.861} C_VEL
LIN {X 0,Y 566.139,Z 235.463,A -85,B 0,C 180,E1 -2391.634,E2 -2391.634} C_VEL
LIN {X 0,Y 566.155,Z 235.46,A -85,B 0,C 180,E1 -2394.308,E2 -2394.308} C_VEL
LIN {X 0,Y 566.171,Z 235.455,A -85,B 0,C 180,E1 -2396.895,E2 -2396.895} C_VEL
LIN {X 0,Y 566.149,Z 235.462,A -85,B 0,C 180,E1 -2399.406,E2 -2399.406} C_VEL
LIN {X 0,Y 566.164,Z 235.463,A -85,B 0,C 180,E1 -2401.856,E2 -2401.856} C_VEL
LIN {X 0,Y 566.167,Z 235.457,A -85,B 0,C 180,E1 -2404.249,E2 -2404.249} C_VEL
LIN {X 0,Y 566.188,Z 235.453,A -85,B 0,C 180,E1 -2406.696,E2 -2406.696} C_VEL
LIN {X 0,Y 566.165,Z 235.463,A -85,B 0,C 180,E1 -2409.662,E2 -2409.662} C_VEL
LIN {X 0,Y 566.194,Z 235.453,A -85,B 0,C 180,E1 -2412.669,E2 -2412.669} C_VEL
LIN {X 0,Y 566.173,Z 235.461,A -85,B 0,C 180,E1 -2415.626,E2 -2415.626} C_VEL
LIN {X 0,Y 566.205,Z 235.453,A -85,B 0,C 180,E1 -2418.652,E2 -2418.652} C_VEL
LIN {X 0,Y 566.199,Z 235.459,A -85,B 0,C 180,E1 -2421.434,E2 -2421.434} C_VEL
LIN {X 0,Y 566.16,Z 235.461,A -85,B 0,C 180,E1 -2423.586,E2 -2423.586} C_VEL
LIN {X 0,Y 566.128,Z 235.463,A -85,B 0,C 180,E1 -2425.728,E2 -2425.728} C_VEL
LIN {X 0,Y 566.211,Z 235.451,A -85,B 0,C 180,E1 -2427.866,E2 -2427.866} C_VEL
LIN {X 0,Y 566.25,Z 235.452,A -85,B 0,C 180,E1 -2430.711,E2 -2430.711} C_VEL
LIN {X 0,Y 566.139,Z 235.461,A -85,B 0,C 180,E1 -2433.559,E2 -2433.559} C_VEL
LIN {X 0,Y 566.203,Z 235.452,A -85,B 0,C 180,E1 -2435.699,E2 -2435.699} C_VEL
LIN {X 0,Y 566.181,Z 235.455,A -85,B 0,C 180,E1 -2437.848,E2 -2437.848} C_VEL
LIN {X 0,Y 566.191,Z 235.462,A -85,B 0,C 180,E1 -2440.73,E2 -2440.73} C_VEL
LIN {X 0,Y 566.15,Z 235.458,A -85,B 0,C 180,E1 -2443.642,E2 -2443.642} C_VEL
LIN {X 0,Y 566.181,Z 235.464,A -85,B 0,C 180,E1 -2446.588,E2 -2446.588} C_VEL
LIN {X 0,Y 566.152,Z 235.457,A -85,B 0,C 180,E1 -2449.582,E2 -2449.582} C_VEL
LIN {X 0,Y 566.165,Z 235.462,A -85,B 0,C 180,E1 -2452.632,E2 -2452.632} C_VEL
LIN {X 0,Y 566.185,Z 235.454,A -85,B 0,C 180,E1 -2455.04,E2 -2455.04} C_VEL
LIN {X 0,Y 566.165,Z 235.455,A -85,B 0,C 180,E1 -2457.341,E2 -2457.341} C_VEL
LIN {X 0,Y 566.182,Z 235.456,A -85,B 0,C 180,E1 -2459.769,E2 -2459.769} C_VEL
LIN {X 0,Y 566.155,Z 235.463,A -85,B 0,C 180,E1 -2462.435,E2 -2462.435} C_VEL
LIN {X 0,Y 566.157,Z 235.457,A -85,B 0,C 180,E1 -2464.998,E2 -2464.998} C_VEL
LIN {X 0,Y 566.144,Z 235.46,A -85,B 0,C 180,E1 -2467.464,E2 -2467.464} C_VEL
LIN {X 0,Y 566.184,Z 235.46,A -85,B 0,C 180,E1 -2470.2,E2 -2470.2} C_VEL
LIN {X 0,Y 566.155,Z 235.457,A -85,B 0,C 180,E1 -2473.057,E2 -2473.057} C_VEL
LIN {X 0,Y 566.179,Z 235.46,A -85,B 0,C 180,E1 -2476.049,E2 -2476.049} C_VEL
LIN {X 0,Y 566.173,Z 235.455,A -85,B 0,C 180,E1 -2478.869,E2 -2478.869} C_VEL
LIN {X 0,Y 566.145,Z 235.467,A -85,B 0,C 180,E1 -2481.642,E2 -2481.642} C_VEL
LIN {X 0,Y 566.17,Z 235.456,A -85,B 0,C 180,E1 -2484.316,E2 -2484.316} C_VEL
LIN {X 0,Y 566.189,Z 235.453,A -85,B 0,C 180,E1 -2486.903,E2 -2486.903} C_VEL
LIN {X 0,Y 566.144,Z 235.466,A -85,B 0,C 180,E1 -2489.412,E2 -2489.412} C_VEL
LIN {X 0,Y 566.192,Z 235.456,A -85,B 0,C 180,E1 -2491.863,E2 -2491.863} C_VEL
LIN {X 0,Y 566.178,Z 235.454,A -85,B 0,C 180,E1 -2494.256,E2 -2494.256} C_VEL
LIN {X 0,Y 566.141,Z 235.46,A -85,B 0,C 180,E1 -2496.723,E2 -2496.723} C_VEL
LIN {X 0,Y 566.19,Z 235.456,A -85,B 0,C 180,E1 -2499.668,E2 -2499.668} C_VEL
LIN {X 0,Y 566.171,Z 235.457,A -85,B 0,C 180,E1 -2502.673,E2 -2502.673} C_VEL
LIN {X 0,Y 566.204,Z 235.453,A -85,B 0,C 180,E1 -2505.631,E2 -2505.631} C_VEL
LIN {X 0,Y 566.256,Z 235.448,A -85,B 0,C 180,E1 -2508.658,E2 -2508.658} C_VEL
LIN {X 0,Y 566.178,Z 235.457,A -85,B 0,C 180,E1 -2511.438,E2 -2511.438} C_VEL
LIN {X 0,Y 566.236,Z 235.448,A -85,B 0,C 180,E1 -2514.306,E2 -2514.306} C_VEL
LIN {X 0,Y 566.25,Z 235.445,A -85,B 0,C 180,E1 -2517.87,E2 -2517.87} C_VEL
LIN {X 0,Y 566.298,Z 235.448,A -85,B 0,C 180,E1 -2520.715,E2 -2520.715} C_VEL
LIN {X 0,Y 566.255,Z 235.452,A -85,B 0,C 180,E1 -2522.85,E2 -2522.85} C_VEL
LIN {X 0,Y 566.231,Z 235.447,A -85,B 0,C 180,E1 -2525.702,E2 -2525.702} C_VEL
LIN {X 0,Y 566.179,Z 235.455,A -85,B 0,C 180,E1 -2527.852,E2 -2527.852} C_VEL
LIN {X 0,Y 566.226,Z 235.454,A -85,B 0,C 180,E1 -2530.733,E2 -2530.733} C_VEL
LIN {X 0,Y 566.183,Z 235.454,A -85,B 0,C 180,E1 -2533.645,E2 -2533.645} C_VEL
LIN {X 0,Y 566.194,Z 235.458,A -85,B 0,C 180,E1 -2536.592,E2 -2536.592} C_VEL
LIN {X 0,Y 566.197,Z 235.452,A -85,B 0,C 180,E1 -2539.584,E2 -2539.584} C_VEL
LIN {X 0,Y 566.189,Z 235.457,A -85,B 0,C 180,E1 -2541.866,E2 -2541.866} C_VEL
LIN {X 0,Y 566.219,Z 235.449,A -85,B 0,C 180,E1 -2545.033,E2 -2545.033} C_VEL
LIN {X 0,Y 566.186,Z 235.461,A -85,B 0,C 180,E1 -2548.201,E2 -2548.201} C_VEL
LIN {X 0,Y 566.185,Z 235.453,A -85,B 0,C 180,E1 -2551.078,E2 -2551.078} C_VEL
LIN {X 0,Y 566.213,Z 235.456,A -85,B 0,C 180,E1 -2553.736,E2 -2553.736} C_VEL
LIN {X 0,Y 566.181,Z 235.455,A -85,B 0,C 180,E1 -2556.574,E2 -2556.574} C_VEL
LIN {X 0,Y 566.212,Z 235.459,A -85,B 0,C 180,E1 -2559.687,E2 -2559.687} C_VEL
LIN {X 0,Y 566.176,Z 235.461,A -85,B 0,C 180,E1 -2562.093,E2 -2562.093} C_VEL
LIN {X 0,Y 566.167,Z 235.462,A -85,B 0,C 180,E1 -2565.039,E2 -2565.039} C_VEL
LIN {X 0,Y 566.26,Z 236.035,A -85,B 0,C 180,E1 -2566.045,E2 -2566.045} C_VEL
LIN {X 0,Y 566.524,Z 239.162,A -85,B 0,C 180,E1 -2568.104,E2 -2568.104} C_VEL
LIN {X 0,Y 566.51,Z 243.529,A -85,B 0,C 180,E1 -2570.752,E2 -2570.752} C_VEL
LIN {X 0,Y 566.41,Z 248.871,A -85,B 0,C 180,E1 -2573.759,E2 -2573.759} C_VEL
LIN {X 0,Y 566.334,Z 253.579,A -85,B 0,C 180,E1 -2576.25,E2 -2576.25} C_VEL
LIN {X 0,Y 566.234,Z 258.243,A -85,B 0,C 180,E1 -2578.582,E2 -2578.582} C_VEL
LIN {X 0,Y 566.143,Z 263.353,A -85,B 0,C 180,E1 -2581.045,E2 -2581.045} C_VEL
LIN {X 0,Y 566.116,Z 268.587,A -85,B 0,C 180,E1 -2583.455,E2 -2583.455} C_VEL
LIN {X 0,Y 566.068,Z 273.848,A -85,B 0,C 180,E1 -2585.814,E2 -2585.814} C_VEL
LIN {X 0,Y 566.04,Z 281.044,A -85,B 0,C 180,E1 -2588.896,E2 -2588.896} C_VEL
LIN {X 0,Y 566.028,Z 286.478,A -85,B 0,C 180,E1 -2591.167,E2 -2591.167} C_VEL
LIN {X 0,Y 565.939,Z 293.664,A -85,B 0,C 180,E1 -2594.145,E2 -2594.145} C_VEL
LIN {X 0,Y 565.938,Z 299.054,A -85,B 0,C 180,E1 -2596.353,E2 -2596.353} C_VEL
LIN {X 0,Y 565.903,Z 301.524,A -85,B 0,C 180,E1 -2597.357,E2 -2597.357} C_VEL
LIN {X 0,Y 566.918,Z 308.476,A -85,B 0,C 180,E1 -2597.516,E2 -2597.516} C_VEL
LIN {X 0,Y 566.798,Z 321.069,A -85,B 0,C 180,E1 -2597.877,E2 -2597.877} C_VEL
LIN {X 0,Y 566.676,Z 331.42,A -85,B 0,C 180,E1 -2598.283,E2 -2598.283} C_VEL
LIN {X 0,Y 566.54,Z 341.634,A -85,B 0,C 180,E1 -2598.795,E2 -2598.795} C_VEL
